LIN {X 0,Y 118.356,Z 1035.076,A -85,B 0,C 180,E1 -26009.999,E2 -26009.999} C_VEL
LIN {X 0,Y 118.425,Z 1040.689,A -85,B 0,C 180,E1 -26012.55,E2 -26012.55} C_VEL
LIN {X 0,Y 118.079,Z 1046.655,A -85,B 0,C 180,E1 -26015.978,E2 -26015.978} C_VEL
LIN {X 0,Y 117.481,Z 1052.345,A -85,B 0,C 180,E1 -26020.338,E2 -26020.338} C_VEL
LIN {X 0,Y 117.718,Z 1057.941,A -85,B 0,C 180,E1 -26025.528,E2 -26025.528} C_VEL
LIN {X 0,Y 119.258,Z 1062.55,A -85,B 0,C 180,E1 -26030.706,E2 -26030.706} C_VEL
LIN {X 0,Y 122.138,Z 1066.32,A -85,B 0,C 180,E1 -26035.566,E2 -26035.566} C_VEL
LIN {X 0,Y 126.034,Z 1069.156,A -85,B 0,C 180,E1 -26040.123,E2 -26040.123} C_VEL
LIN {X 0,Y 129.271,Z 1070.735,A -85,B 0,C 180,E1 -26042.933,E2 -26042.933} C_VEL
LIN {X 0,Y 137.158,Z 1072.698,A -85,B 0,C 180,E1 -26047.943,E2 -26047.943} C_VEL
LIN {X 0,Y 141.648,Z 1073.261,A -85,B 0,C 180,E1 -26050.166,E2 -26050.166} C_VEL
LIN {X 0,Y 151.624,Z 1073.236,A -85,B 0,C 180,E1 -26054.048,E2 -26054.048} C_VEL
LIN {X 0,Y 157.044,Z 1072.693,A -85,B 0,C 180,E1 -26055.727,E2 -26055.727} C_VEL
LIN {X 0,Y 157.853,Z 1072.521,A -85,B 0,C 180,E1 -26056.542,E2 -26056.542} C_VEL
LIN {X 0,Y 150.11,Z 1072.526,A -85,B 0,C 180,E1 -26059.047,E2 -26059.047} C_VEL
LIN {X 0,Y 142.602,Z 1071.645,A -85,B 0,C 180,E1 -26062.049,E2 -26062.049} C_VEL
LIN {X 0,Y 135.958,Z 1069.937,A -85,B 0,C 180,E1 -26065.348,E2 -26065.348} C_VEL
LIN {X 0,Y 130,Z 1067.367,A -85,B 0,C 180,E1 -26069.099,E2 -26069.099} C_VEL
LIN {X 0,Y 124.977,Z 1063.891,A -85,B 0,C 180,E1 -26073.266,E2 -26073.266} C_VEL
LIN {X 0,Y 121.04,Z 1059.399,A -85,B 0,C 180,E1 -26078.008,E2 -26078.008} C_VEL
LIN {X 0,Y 117.924,Z 1053.086,A -85,B 0,C 180,E1 -26083.593,E2 -26083.593} C_VEL
LIN {X 0,Y 116.582,Z 1047.62,A -85,B 0,C 180,E1 -26087.821,E2 -26087.821} C_VEL
LIN {X 0,Y 116.174,Z 1041.128,A -85,B 0,C 180,E1 -26092.179,E2 -26092.179} C_VEL
LIN {X 0,Y 116.121,Z 1034.894,A -85,B 0,C 180,E1 -26095.709,E2 -26095.709} C_VEL
LIN {X 0,Y 115.59,Z 1030.657,A -85,B 0,C 180,E1 -26097.651,E2 -26097.651} C_VEL
LIN {X 0,Y 114.297,Z 1025.939,A -85,B 0,C 180,E1 -26099.273,E2 -26099.273} C_VEL
LIN {X 0,Y 110.803,Z 1013.931,A -85,B 0,C 180,E1 -26102.592,E2 -26102.592} C_VEL
LIN {X 0,Y 110.37,Z 1008.52,A -85,B 0,C 180,E1 -26104.089,E2 -26104.089} C_VEL
LIN {X 0,Y 110.83,Z 996.455,A -85,B 0,C 180,E1 -26107.059,E2 -26107.059} C_VEL
LIN {X 0,Y 111.232,Z 984.797,A -85,B 0,C 180,E1 -26109.205,E2 -26109.205} C_VEL
LIN {X 0,Y 111.564,Z 944.315,A -85,B 0,C 180,E1 -26114.869,E2 -26114.869} C_VEL
LIN {X 0,Y 111.563,Z 935.848,A -85,B 0,C 180,E1 -26115.986,E2 -26115.986} C_VEL
LIN {X 0,Y 109.071,Z 921.711,A -85,B 0,C 180,E1 -26117.593,E2 -26117.593} C_VEL
LIN {X 0,Y 107.833,Z 921.864,A -85,B 0,C 180,E1 -26127.146,E2 -26127.146} C_VEL
LIN {X 0,Y 107.78,Z 921.869,A -85,B 0,C 180,E1 -26132.039,E2 -26132.039} C_VEL
LIN {X 0,Y 107.684,Z 921.876,A -85,B 0,C 180,E1 -26138.448,E2 -26138.448} C_VEL
LIN {X 0,Y 107.671,Z 921.883,A -85,B 0,C 180,E1 -26145.893,E2 -26145.893} C_VEL
LIN {X 0,Y 107.685,Z 921.882,A -85,B 0,C 180,E1 -26151.555,E2 -26151.555} C_VEL
LIN {X 0,Y 107.793,Z 921.862,A -85,B 0,C 180,E1 -26158.562,E2 -26158.562} C_VEL
LIN {X 0,Y 107.882,Z 921.851,A -85,B 0,C 180,E1 -26166.992,E2 -26166.992} C_VEL
LIN {X 0,Y 107.973,Z 921.842,A -85,B 0,C 180,E1 -26174.909,E2 -26174.909} C_VEL
LIN {X 0,Y 108.23,Z 921.813,A -85,B 0,C 180,E1 -26178.767,E2 -26178.767} C_VEL
LIN {X 0,Y 108.291,Z 921.806,A -85,B 0,C 180,E1 -26182.543,E2 -26182.543} C_VEL
LIN {X 0,Y 108.876,Z 921.737,A -85,B 0,C 180,E1 -26190.001,E2 -26190.001} C_VEL
LIN {X 0,Y 108.291,Z 921.806,A -85,B 0,C 180,E1 -26197.459,E2 -26197.459} C_VEL
LIN {X 0,Y 108.142,Z 921.819,A -85,B 0,C 180,E1 -26202.874,E2 -26202.874} C_VEL
LIN {X 0,Y 107.863,Z 921.862,A -85,B 0,C 180,E1 -26209.014,E2 -26209.014} C_VEL
LIN {X 0,Y 107.806,Z 921.862,A -85,B 0,C 180,E1 -26214.117,E2 -26214.117} C_VEL
LIN {X 0,Y 107.776,Z 921.863,A -85,B 0,C 180,E1 -26222.032,E2 -26222.032} C_VEL
LIN {X 0,Y 107.687,Z 921.882,A -85,B 0,C 180,E1 -26228.446,E2 -26228.446} C_VEL
LIN {X 0,Y 107.673,Z 921.886,A -85,B 0,C 180,E1 -26235.89,E2 -26235.89} C_VEL
LIN {X 0,Y 107.686,Z 921.876,A -85,B 0,C 180,E1 -26241.553,E2 -26241.553} C_VEL
LIN {X 0,Y 107.787,Z 921.865,A -85,B 0,C 180,E1 -26248.557,E2 -26248.557} C_VEL
LIN {X 0,Y 107.869,Z 921.857,A -85,B 0,C 180,E1 -26256.986,E2 -26256.986} C_VEL
LIN {X 0,Y 107.863,Z 921.856,A -85,B 0,C 180,E1 -26260.985,E2 -26260.985} C_VEL
LIN {X 0,Y 108.209,Z 921.809,A -85,B 0,C 180,E1 -26268.763,E2 -26268.763} C_VEL
LIN {X 0,Y 108.289,Z 921.808,A -85,B 0,C 180,E1 -26272.54,E2 -26272.54} C_VEL
LIN {X 0,Y 108.873,Z 921.732,A -85,B 0,C 180,E1 -26279.998,E2 -26279.998} C_VEL
LIN {X 0,Y 108.284,Z 921.801,A -85,B 0,C 180,E1 -26287.457,E2 -26287.457} C_VEL
LIN {X 0,Y 108.138,Z 921.826,A -85,B 0,C 180,E1 -26292.87,E2 -26292.87} C_VEL
LIN {X 0,Y 107.861,Z 921.86,A -85,B 0,C 180,E1 -26299.012,E2 -26299.012} C_VEL
LIN {X 0,Y 107.802,Z 921.864,A -85,B 0,C 180,E1 -26304.115,E2 -26304.115} C_VEL
LIN {X 0,Y 107.772,Z 921.87,A -85,B 0,C 180,E1 -26312.031,E2 -26312.031} C_VEL
LIN {X 0,Y 107.683,Z 921.883,A -85,B 0,C 180,E1 -26318.445,E2 -26318.445} C_VEL
LIN {X 0,Y 107.668,Z 921.882,A -85,B 0,C 180,E1 -26325.889,E2 -26325.889} C_VEL
LIN {X 0,Y 107.69,Z 921.879,A -85,B 0,C 180,E1 -26331.546,E2 -26331.546} C_VEL
LIN {X 0,Y 108.007,Z 921.843,A -85,B 0,C 180,E1 -26338.629,E2 -26338.629} C_VEL
LIN {X 0,Y 108.535,Z 921.78,A -85,B 0,C 180,E1 -26345.029,E2 -26345.029} C_VEL
LIN {X 0,Y 108.52,Z 921.977,A -85,B 0,C 180,E1 -26351.306,E2 -26351.306} C_VEL
LIN {X 0,Y 109.506,Z 943.925,A -85,B 0,C 180,E1 -26354.093,E2 -26354.093} C_VEL
LIN {X 0,Y 111.954,Z 966.951,A -85,B 0,C 180,E1 -26356.846,E2 -26356.846} C_VEL
LIN {X 0,Y 112.053,Z 995.999,A -85,B 0,C 180,E1 -26360.978,E2 -26360.978} C_VEL
LIN {X 0,Y 111.956,Z 1007.75,A -85,B 0,C 180,E1 -26363.24,E2 -26363.24} C_VEL
LIN {X 0,Y 111.912,Z 1018.14,A -85,B 0,C 180,E1 -26365.948,E2 -26365.948} C_VEL
LIN {X 0,Y 111.98,Z 1027.568,A -85,B 0,C 180,E1 -26369.1,E2 -26369.1} C_VEL
LIN {X 0,Y 112.088,Z 1034.186,A -85,B 0,C 180,E1 -26371.796,E2 -26371.796} C_VEL
LIN {X 0,Y 112.177,Z 1039.691,A -85,B 0,C 180,E1 -26374.491,E2 -26374.491} C_VEL
LIN {X 0,Y 111.753,Z 1045.35,A -85,B 0,C 180,E1 -26378.134,E2 -26378.134} C_VEL
LIN {X 0,Y 111.322,Z 1051.047,A -85,B 0,C 180,E1 -26382.765,E2 -26382.765} C_VEL
LIN {X 0,Y 112.15,Z 1057.246,A -85,B 0,C 180,E1 -26389.015,E2 -26389.015} C_VEL
LIN {X 0,Y 114.029,Z 1061.308,A -85,B 0,C 180,E1 -26393.616,E2 -26393.616} C_VEL
LIN {X 0,Y 117.42,Z 1065.087,A -85,B 0,C 180,E1 -26398.608,E2 -26398.608} C_VEL
LIN {X 0,Y 120.205,Z 1067.17,A -85,B 0,C 180,E1 -26401.749,E2 -26401.749} C_VEL
LIN {X 0,Y 127.45,Z 1070.367,A -85,B 0,C 180,E1 -26407.342,E2 -26407.342} C_VEL
LIN {X 0,Y 136.354,Z 1072.23,A -85,B 0,C 180,E1 -26412.07,E2 -26412.07} C_VEL
LIN {X 0,Y 141.307,Z 1072.763,A -85,B 0,C 180,E1 -26414.13,E2 -26414.13} C_VEL
LIN {X 0,Y 146.601,Z 1072.841,A -85,B 0,C 180,E1 -26415.979,E2 -26415.979} C_VEL
LIN {X 0,Y 144.811,Z 1072.568,A -85,B 0,C 180,E1 -26417.201,E2 -26417.201} C_VEL
LIN {X 0,Y 134.801,Z 1070.653,A -85,B 0,C 180,E1 -26421.273,E2 -26421.273} C_VEL
LIN {X 0,Y 126.016,Z 1067.11,A -85,B 0,C 180,E1 -26426.104,E2 -26426.104} C_VEL
LIN {X 0,Y 120.483,Z 1063.528,A -85,B 0,C 180,E1 -26430.278,E2 -26430.278} C_VEL
LIN {X 0,Y 116.099,Z 1059.034,A -85,B 0,C 180,E1 -26434.931,E2 -26434.931} C_VEL
LIN {X 0,Y 113.167,Z 1054.345,A -85,B 0,C 180,E1 -26439.358,E2 -26439.358} C_VEL
LIN {X 0,Y 110.941,Z 1048.163,A -85,B 0,C 180,E1 -26444.383,E2 -26444.383} C_VEL
LIN {X 0,Y 109.917,Z 1040.561,A -85,B 0,C 180,E1 -26449.875,E2 -26449.875} C_VEL
LIN {X 0,Y 109.813,Z 1032.534,A -85,B 0,C 180,E1 -26454.6,E2 -26454.6} C_VEL
LIN {X 0,Y 109.86,Z 1024.026,A -85,B 0,C 180,E1 -26458.627,E2 -26458.627} C_VEL
LIN {X 0,Y 110.115,Z 1014.241,A -85,B 0,C 180,E1 -26462.288,E2 -26462.288} C_VEL
LIN {X 0,Y 110.37,Z 1008.52,A -85,B 0,C 180,E1 -26464.089,E2 -26464.089} C_VEL
LIN {X 0,Y 109.99,Z 1003.267,A -85,B 0,C 180,E1 -26465.388,E2 -26465.388} C_VEL
LIN {X 0,Y 108.798,Z 997.812,A -85,B 0,C 180,E1 -26466.343,E2 -26466.343} C_VEL
LIN {X 0,Y 104.989,Z 982.527,A -85,B 0,C 180,E1 -26468.19,E2 -26468.19} C_VEL
LIN {X 0,Y 104.586,Z 978.592,A -85,B 0,C 180,E1 -26468.697,E2 -26468.697} C_VEL
LIN {X 0,Y 104.815,Z 939.202,A -85,B 0,C 180,E1 -26474.565,E2 -26474.565} C_VEL
LIN {X 0,Y 104.403,Z 933.942,A -85,B 0,C 180,E1 -26475.247,E2 -26475.247} C_VEL
LIN {X 0,Y 102.249,Z 922.562,A -85,B 0,C 180,E1 -26476.614,E2 -26476.614} C_VEL
LIN {X 0,Y 100.884,Z 922.732,A -85,B 0,C 180,E1 -26485.092,E2 -26485.092} C_VEL
LIN {X 0,Y 100.689,Z 922.753,A -85,B 0,C 180,E1 -26493.114,E2 -26493.114} C_VEL
LIN {X 0,Y 100.635,Z 922.753,A -85,B 0,C 180,E1 -26499.809,E2 -26499.809} C_VEL
LIN {X 0,Y 100.642,Z 922.759,A -85,B 0,C 180,E1 -26505.709,E2 -26505.709} C_VEL
LIN {X 0,Y 100.623,Z 922.762,A -85,B 0,C 180,E1 -26511.054,E2 -26511.054} C_VEL
LIN {X 0,Y 100.69,Z 922.746,A -85,B 0,C 180,E1 -26516.889,E2 -26516.889} C_VEL
LIN {X 0,Y 100.737,Z 922.744,A -85,B 0,C 180,E1 -26525.093,E2 -26525.093} C_VEL
LIN {X 0,Y 100.785,Z 922.742,A -85,B 0,C 180,E1 -26529.595,E2 -26529.595} C_VEL
LIN {X 0,Y 101.129,Z 922.696,A -85,B 0,C 180,E1 -26537.967,E2 -26537.967} C_VEL
LIN {X 0,Y 101.229,Z 922.687,A -85,B 0,C 180,E1 -26542.019,E2 -26542.019} C_VEL
LIN {X 0,Y 101.807,Z 922.617,A -85,B 0,C 180,E1 -26550.001,E2 -26550.001} C_VEL
LIN {X 0,Y 101.228,Z 922.687,A -85,B 0,C 180,E1 -26557.982,E2 -26557.982} C_VEL
LIN {X 0,Y 101.054,Z 922.701,A -85,B 0,C 180,E1 -26563.171,E2 -26563.171} C_VEL
LIN {X 0,Y 100.777,Z 922.743,A -85,B 0,C 180,E1 -26570.408,E2 -26570.408} C_VEL
LIN {X 0,Y 100.721,Z 922.746,A -85,B 0,C 180,E1 -26574.887,E2 -26574.887} C_VEL
LIN {X 0,Y 100.688,Z 922.747,A -85,B 0,C 180,E1 -26583.109,E2 -26583.109} C_VEL
LIN {X 0,Y 100.638,Z 922.756,A -85,B 0,C 180,E1 -26589.806,E2 -26589.806} C_VEL
LIN {X 0,Y 100.644,Z 922.761,A -85,B 0,C 180,E1 -26595.706,E2 -26595.706} C_VEL
LIN {X 0,Y 100.624,Z 922.754,A -85,B 0,C 180,E1 -26601.051,E2 -26601.051} C_VEL
LIN {X 0,Y 100.688,Z 922.754,A -85,B 0,C 180,E1 -26606.889,E2 -26606.889} C_VEL
LIN {X 0,Y 100.745,Z 922.748,A -85,B 0,C 180,E1 -26615.254,E2 -26615.254} C_VEL
LIN {X 0,Y 100.778,Z 922.736,A -85,B 0,C 180,E1 -26619.591,E2 -26619.591} C_VEL
LIN {X 0,Y 101.118,Z 922.692,A -85,B 0,C 180,E1 -26627.963,E2 -26627.963} C_VEL
LIN {X 0,Y 101.224,Z 922.689,A -85,B 0,C 180,E1 -26632.016,E2 -26632.016} C_VEL
LIN {X 0,Y 101.805,Z 922.613,A -85,B 0,C 180,E1 -26639.998,E2 -26639.998} C_VEL
LIN {X 0,Y 101.219,Z 922.681,A -85,B 0,C 180,E1 -26647.98,E2 -26647.98} C_VEL
LIN {X 0,Y 101.051,Z 922.708,A -85,B 0,C 180,E1 -26653.169,E2 -26653.169} C_VEL
LIN {X 0,Y 100.774,Z 922.744,A -85,B 0,C 180,E1 -26660.406,E2 -26660.406} C_VEL
LIN {X 0,Y 100.717,Z 922.743,A -85,B 0,C 180,E1 -26664.886,E2 -26664.886} C_VEL
LIN {X 0,Y 100.684,Z 922.75,A -85,B 0,C 180,E1 -26673.108,E2 -26673.108} C_VEL
LIN {X 0,Y 100.634,Z 922.762,A -85,B 0,C 180,E1 -26679.805,E2 -26679.805} C_VEL
LIN {X 0,Y 100.639,Z 922.756,A -85,B 0,C 180,E1 -26685.705,E2 -26685.705} C_VEL
LIN {X 0,Y 100.627,Z 922.759,A -85,B 0,C 180,E1 -26691.054,E2 -26691.054} C_VEL
LIN {X 0,Y 100.793,Z 922.743,A -85,B 0,C 180,E1 -26696.793,E2 -26696.793} C_VEL
LIN {X 0,Y 101.378,Z 922.668,A -85,B 0,C 180,E1 -26704.315,E2 -26704.315} C_VEL
LIN {X 0,Y 101.61,Z 922.642,A -85,B 0,C 180,E1 -26712.255,E2 -26712.255} C_VEL
LIN {X 0,Y 102.806,Z 945.114,A -85,B 0,C 180,E1 -26715.335,E2 -26715.335} C_VEL
LIN {X 0,Y 105.267,Z 967.587,A -85,B 0,C 180,E1 -26718.201,E2 -26718.201} C_VEL
LIN {X 0,Y 105.553,Z 996.226,A -85,B 0,C 180,E1 -26722.587,E2 -26722.587} C_VEL
LIN {X 0,Y 105.558,Z 1008.784,A -85,B 0,C 180,E1 -26725.225,E2 -26725.225} C_VEL
LIN {X 0,Y 105.625,Z 1020.086,A -85,B 0,C 180,E1 -26728.568,E2 -26728.568} C_VEL
LIN {X 0,Y 105.891,Z 1028.857,A -85,B 0,C 180,E1 -26731.901,E2 -26731.901} C_VEL
LIN {X 0,Y 106.139,Z 1036.77,A -85,B 0,C 180,E1 -26735.701,E2 -26735.701} C_VEL
LIN {X 0,Y 105.886,Z 1041.269,A -85,B 0,C 180,E1 -26738.588,E2 -26738.588} C_VEL
LIN {X 0,Y 105.412,Z 1047.304,A -85,B 0,C 180,E1 -26743.494,E2 -26743.494} C_VEL
LIN {X 0,Y 106.318,Z 1054.567,A -85,B 0,C 180,E1 -26750.676,E2 -26750.676} C_VEL
LIN {X 0,Y 110.355,Z 1061.207,A -85,B 0,C 180,E1 -26758.531,E2 -26758.531} C_VEL
LIN {X 0,Y 114.566,Z 1064.808,A -85,B 0,C 180,E1 -26763.511,E2 -26763.511} C_VEL
LIN {X 0,Y 118.065,Z 1066.85,A -85,B 0,C 180,E1 -26766.531,E2 -26766.531} C_VEL
LIN {X 0,Y 126.486,Z 1069.936,A -85,B 0,C 180,E1 -26771.817,E2 -26771.817} C_VEL
LIN {X 0,Y 136.365,Z 1071.739,A -85,B 0,C 180,E1 -26776.181,E2 -26776.181} C_VEL
LIN {X 0,Y 132.956,Z 1070.914,A -85,B 0,C 180,E1 -26777.734,E2 -26777.734} C_VEL
LIN {X 0,Y 122.436,Z 1066.822,A -85,B 0,C 180,E1 -26782.937,E2 -26782.937} C_VEL
LIN {X 0,Y 116.375,Z 1063.037,A -85,B 0,C 180,E1 -26787.078,E2 -26787.078} C_VEL
LIN {X 0,Y 111.285,Z 1058.298,A -85,B 0,C 180,E1 -26791.936,E2 -26791.936} C_VEL
LIN {X 0,Y 107.022,Z 1051.645,A -85,B 0,C 180,E1 -26798.114,E2 -26798.114} C_VEL
LIN {X 0,Y 104.467,Z 1043.763,A -85,B 0,C 180,E1 -26804.391,E2 -26804.391} C_VEL
LIN {X 0,Y 103.735,Z 1035.281,A -85,B 0,C 180,E1 -26810.25,E2 -26810.25} C_VEL
LIN {X 0,Y 103.661,Z 1028.425,A -85,B 0,C 180,E1 -26814.165,E2 -26814.165} C_VEL
LIN {X 0,Y 103.678,Z 1019.9,A -85,B 0,C 180,E1 -26818.059,E2 -26818.059} C_VEL
LIN {X 0,Y 103.888,Z 1009.362,A -85,B 0,C 180,E1 -26821.94,E2 -26821.94} C_VEL
LIN {X 0,Y 104.223,Z 998.058,A -85,B 0,C 180,E1 -26825.079,E2 -26825.079} C_VEL
LIN {X 0,Y 104.551,Z 987.696,A -85,B 0,C 180,E1 -26827.243,E2 -26827.243} C_VEL
LIN {X 0,Y 104.586,Z 978.592,A -85,B 0,C 180,E1 -26828.697,E2 -26828.697} C_VEL
LIN {X 0,Y 103.841,Z 972.861,A -85,B 0,C 180,E1 -26829.409,E2 -26829.409} C_VEL
LIN {X 0,Y 98.573,Z 954.007,A -85,B 0,C 180,E1 -26831.225,E2 -26831.225} C_VEL
LIN {X 0,Y 97.979,Z 948.282,A -85,B 0,C 180,E1 -26832.006,E2 -26832.006} C_VEL
LIN {X 0,Y 97.787,Z 935.443,A -85,B 0,C 180,E1 -26833.957,E2 -26833.957} C_VEL
LIN {X 0,Y 95.48,Z 923.405,A -85,B 0,C 180,E1 -26835.453,E2 -26835.453} C_VEL
LIN {X 0,Y 93.708,Z 923.625,A -85,B 0,C 180,E1 -26846.746,E2 -26846.746} C_VEL
LIN {X 0,Y 93.585,Z 923.64,A -85,B 0,C 180,E1 -26854.304,E2 -26854.304} C_VEL
LIN {X 0,Y 93.529,Z 923.647,A -85,B 0,C 180,E1 -26862.557,E2 -26862.557} C_VEL
LIN {X 0,Y 93.532,Z 923.638,A -85,B 0,C 180,E1 -26868.715,E2 -26868.715} C_VEL
LIN {X 0,Y 93.586,Z 923.636,A -85,B 0,C 180,E1 -26875.7,E2 -26875.7} C_VEL
LIN {X 0,Y 93.646,Z 923.631,A -85,B 0,C 180,E1 -26884.24,E2 -26884.24} C_VEL
LIN {X 0,Y 93.657,Z 923.624,A -85,B 0,C 180,E1 -26887.964,E2 -26887.964} C_VEL
LIN {X 0,Y 94.019,Z 923.577,A -85,B 0,C 180,E1 -26897.042,E2 -26897.042} C_VEL
LIN {X 0,Y 94.16,Z 923.569,A -85,B 0,C 180,E1 -26901.416,E2 -26901.416} C_VEL
LIN {X 0,Y 94.739,Z 923.497,A -85,B 0,C 180,E1 -26910.001,E2 -26910.001} C_VEL
LIN {X 0,Y 94.16,Z 923.569,A -85,B 0,C 180,E1 -26918.586,E2 -26918.586} C_VEL
LIN {X 0,Y 93.962,Z 923.584,A -85,B 0,C 180,E1 -26923.496,E2 -26923.496} C_VEL
LIN {X 0,Y 93.646,Z 923.625,A -85,B 0,C 180,E1 -26932.04,E2 -26932.04} C_VEL
LIN {X 0,Y 93.591,Z 923.639,A -85,B 0,C 180,E1 -26936.78,E2 -26936.78} C_VEL
LIN {X 0,Y 93.586,Z 923.636,A -85,B 0,C 180,E1 -26944.299,E2 -26944.299} C_VEL
LIN {X 0,Y 93.531,Z 923.64,A -85,B 0,C 180,E1 -26952.554,E2 -26952.554} C_VEL
LIN {X 0,Y 93.534,Z 923.642,A -85,B 0,C 180,E1 -26958.712,E2 -26958.712} C_VEL
LIN {X 0,Y 93.585,Z 923.64,A -85,B 0,C 180,E1 -26965.699,E2 -26965.699} C_VEL
LIN {X 0,Y 93.644,Z 923.632,A -85,B 0,C 180,E1 -26974.239,E2 -26974.239} C_VEL
LIN {X 0,Y 93.653,Z 923.625,A -85,B 0,C 180,E1 -26977.96,E2 -26977.96} C_VEL
LIN {X 0,Y 94.018,Z 923.58,A -85,B 0,C 180,E1 -26987.039,E2 -26987.039} C_VEL
LIN {X 0,Y 94.135,Z 923.57,A -85,B 0,C 180,E1 -26991.411,E2 -26991.411} C_VEL
LIN {X 0,Y 94.737,Z 923.493,A -85,B 0,C 180,E1 -26999.998,E2 -26999.998} C_VEL
LIN {X 0,Y 94.131,Z 923.566,A -85,B 0,C 180,E1 -27008.586,E2 -27008.586} C_VEL
LIN {X 0,Y 93.959,Z 923.591,A -85,B 0,C 180,E1 -27013.494,E2 -27013.494} C_VEL
LIN {X 0,Y 93.643,Z 923.632,A -85,B 0,C 180,E1 -27022.038,E2 -27022.038} C_VEL
LIN {X 0,Y 93.587,Z 923.633,A -85,B 0,C 180,E1 -27026.779,E2 -27026.779} C_VEL
LIN {X 0,Y 93.582,Z 923.63,A -85,B 0,C 180,E1 -27034.298,E2 -27034.298} C_VEL
LIN {X 0,Y 93.526,Z 923.641,A -85,B 0,C 180,E1 -27042.553,E2 -27042.553} C_VEL
LIN {X 0,Y 93.532,Z 923.646,A -85,B 0,C 180,E1 -27048.709,E2 -27048.709} C_VEL
LIN {X 0,Y 93.655,Z 923.629,A -85,B 0,C 180,E1 -27055.632,E2 -27055.632} C_VEL
LIN {X 0,Y 94.206,Z 923.556,A -85,B 0,C 180,E1 -27063.534,E2 -27063.534} C_VEL
LIN {X 0,Y 94.314,Z 923.55,A -85,B 0,C 180,E1 -27068.124,E2 -27068.124} C_VEL
LIN {X 0,Y 94.794,Z 923.492,A -85,B 0,C 180,E1 -27073.436,E2 -27073.436} C_VEL
LIN {X 0,Y 96.131,Z 945.61,A -85,B 0,C 180,E1 -27076.686,E2 -27076.686} C_VEL
LIN {X 0,Y 98.642,Z 967.237,A -85,B 0,C 180,E1 -27079.609,E2 -27079.609} C_VEL
LIN {X 0,Y 99.15,Z 995.476,A -85,B 0,C 180,E1 -27084.253,E2 -27084.253} C_VEL
LIN {X 0,Y 99.307,Z 1007.466,A -85,B 0,C 180,E1 -27086.957,E2 -27086.957} C_VEL
LIN {X 0,Y 99.531,Z 1018.258,A -85,B 0,C 180,E1 -27090.32,E2 -27090.32} C_VEL
LIN {X 0,Y 99.883,Z 1026.452,A -85,B 0,C 180,E1 -27093.529,E2 -27093.529} C_VEL
LIN {X 0,Y 100.183,Z 1033.301,A -85,B 0,C 180,E1 -27096.848,E2 -27096.848} C_VEL
LIN {X 0,Y 99.959,Z 1038.433,A -85,B 0,C 180,E1 -27100.169,E2 -27100.169} C_VEL
LIN {X 0,Y 99.7,Z 1045.625,A -85,B 0,C 180,E1 -27106.377,E2 -27106.377} C_VEL
LIN {X 0,Y 100.786,Z 1051.611,A -85,B 0,C 180,E1 -27112.552,E2 -27112.552} C_VEL
LIN {X 0,Y 103.506,Z 1056.729,A -85,B 0,C 180,E1 -27118.378,E2 -27118.378} C_VEL
LIN {X 0,Y 107.553,Z 1060.954,A -85,B 0,C 180,E1 -27123.74,E2 -27123.74} C_VEL
LIN {X 0,Y 112.777,Z 1064.465,A -85,B 0,C 180,E1 -27128.548,E2 -27128.548} C_VEL
LIN {X 0,Y 116.911,Z 1066.461,A -85,B 0,C 180,E1 -27131.395,E2 -27131.395} C_VEL
LIN {X 0,Y 124.966,Z 1069.131,A -85,B 0,C 180,E1 -27135.675,E2 -27135.675} C_VEL
LIN {X 0,Y 125.191,Z 1069.057,A -85,B 0,C 180,E1 -27136.721,E2 -27136.721} C_VEL
LIN {X 0,Y 116.982,Z 1065.239,A -85,B 0,C 180,E1 -27140.892,E2 -27140.892} C_VEL
LIN {X 0,Y 110.708,Z 1061.033,A -85,B 0,C 180,E1 -27145.158,E2 -27145.158} C_VEL
LIN {X 0,Y 105.602,Z 1055.984,A -85,B 0,C 180,E1 -27150.057,E2 -27150.057} C_VEL
LIN {X 0,Y 101.72,Z 1049.995,A -85,B 0,C 180,E1 -27155.511,E2 -27155.511} C_VEL
LIN {X 0,Y 99.018,Z 1042.801,A -85,B 0,C 180,E1 -27161.376,E2 -27161.376} C_VEL
LIN {X 0,Y 97.939,Z 1035.838,A -85,B 0,C 180,E1 -27166.515,E2 -27166.515} C_VEL
LIN {X 0,Y 97.656,Z 1029.281,A -85,B 0,C 180,E1 -27170.683,E2 -27170.683} C_VEL
LIN {X 0,Y 97.563,Z 1022.495,A -85,B 0,C 180,E1 -27174.317,E2 -27174.317} C_VEL
LIN {X 0,Y 97.56,Z 1014.148,A -85,B 0,C 180,E1 -27177.938,E2 -27177.938} C_VEL
LIN {X 0,Y 97.702,Z 1003.575,A -85,B 0,C 180,E1 -27181.548,E2 -27181.548} C_VEL
LIN {X 0,Y 97.991,Z 991.655,A -85,B 0,C 180,E1 -27184.63,E2 -27184.63} C_VEL
LIN {X 0,Y 98.148,Z 980.058,A -85,B 0,C 180,E1 -27186.813,E2 -27186.813} C_VEL
LIN {X 0,Y 97.979,Z 948.282,A -85,B 0,C 180,E1 -27192.006,E2 -27192.006} C_VEL
LIN {X 0,Y 97.305,Z 944.486,A -85,B 0,C 180,E1 -27192.478,E2 -27192.478} C_VEL
LIN {X 0,Y 94.335,Z 938.527,A -85,B 0,C 180,E1 -27192.8,E2 -27192.8} C_VEL
LIN {X 0,Y 90.979,Z 932.584,A -85,B 0,C 180,E1 -27193.04,E2 -27193.04} C_VEL
LIN {X 0,Y 89.737,Z 928.775,A -85,B 0,C 180,E1 -27193.406,E2 -27193.406} C_VEL
LIN {X 0,Y 88.817,Z 924.232,A -85,B 0,C 180,E1 -27194.044,E2 -27194.044} C_VEL
LIN {X 0,Y 86.54,Z 924.509,A -85,B 0,C 180,E1 -27209.164,E2 -27209.164} C_VEL
LIN {X 0,Y 86.503,Z 924.521,A -85,B 0,C 180,E1 -27215.665,E2 -27215.665} C_VEL
LIN {X 0,Y 86.473,Z 924.525,A -85,B 0,C 180,E1 -27222.992,E2 -27222.992} C_VEL
LIN {X 0,Y 86.455,Z 924.52,A -85,B 0,C 180,E1 -27229.435,E2 -27229.435} C_VEL
LIN {X 0,Y 86.529,Z 924.516,A -85,B 0,C 180,E1 -27235.352,E2 -27235.352} C_VEL
LIN {X 0,Y 86.569,Z 924.513,A -85,B 0,C 180,E1 -27243.261,E2 -27243.261} C_VEL
LIN {X 0,Y 86.603,Z 924.51,A -85,B 0,C 180,E1 -27251.059,E2 -27251.059} C_VEL
LIN {X 0,Y 86.866,Z 924.467,A -85,B 0,C 180,E1 -27256.147,E2 -27256.147} C_VEL
LIN {X 0,Y 87.064,Z 924.452,A -85,B 0,C 180,E1 -27260.71,E2 -27260.71} C_VEL
LIN {X 0,Y 87.672,Z 924.378,A -85,B 0,C 180,E1 -27270.001,E2 -27270.001} C_VEL
LIN {X 0,Y 87.063,Z 924.452,A -85,B 0,C 180,E1 -27279.292,E2 -27279.292} C_VEL
LIN {X 0,Y 86.863,Z 924.467,A -85,B 0,C 180,E1 -27284.048,E2 -27284.048} C_VEL
LIN {X 0,Y 86.597,Z 924.511,A -85,B 0,C 180,E1 -27288.944,E2 -27288.944} C_VEL
LIN {X 0,Y 86.559,Z 924.514,A -85,B 0,C 180,E1 -27296.726,E2 -27296.726} C_VEL
LIN {X 0,Y 86.505,Z 924.521,A -85,B 0,C 180,E1 -27305.661,E2 -27305.661} C_VEL
LIN {X 0,Y 86.475,Z 924.52,A -85,B 0,C 180,E1 -27312.989,E2 -27312.989} C_VEL
LIN {X 0,Y 86.456,Z 924.521,A -85,B 0,C 180,E1 -27319.431,E2 -27319.431} C_VEL
LIN {X 0,Y 86.529,Z 924.519,A -85,B 0,C 180,E1 -27325.348,E2 -27325.348} C_VEL
LIN {X 0,Y 86.565,Z 924.514,A -85,B 0,C 180,E1 -27333.263,E2 -27333.263} C_VEL
LIN {X 0,Y 86.598,Z 924.505,A -85,B 0,C 180,E1 -27341.055,E2 -27341.055} C_VEL
LIN {X 0,Y 86.864,Z 924.474,A -85,B 0,C 180,E1 -27346.147,E2 -27346.147} C_VEL
LIN {X 0,Y 87.028,Z 924.454,A -85,B 0,C 180,E1 -27350.703,E2 -27350.703} C_VEL
LIN {X 0,Y 87.669,Z 924.373,A -85,B 0,C 180,E1 -27359.998,E2 -27359.998} C_VEL
LIN {X 0,Y 87.025,Z 924.455,A -85,B 0,C 180,E1 -27369.293,E2 -27369.293} C_VEL
LIN {X 0,Y 86.86,Z 924.474,A -85,B 0,C 180,E1 -27374.046,E2 -27374.046} C_VEL
LIN {X 0,Y 86.594,Z 924.509,A -85,B 0,C 180,E1 -27378.942,E2 -27378.942} C_VEL
LIN {X 0,Y 86.555,Z 924.509,A -85,B 0,C 180,E1 -27386.724,E2 -27386.724} C_VEL
LIN {X 0,Y 86.501,Z 924.514,A -85,B 0,C 180,E1 -27395.659,E2 -27395.659} C_VEL
LIN {X 0,Y 86.45,Z 924.521,A -85,B 0,C 180,E1 -27402.973,E2 -27402.973} C_VEL
LIN {X 0,Y 86.458,Z 924.527,A -85,B 0,C 180,E1 -27409.434,E2 -27409.434} C_VEL
LIN {X 0,Y 86.59,Z 924.509,A -85,B 0,C 180,E1 -27415.378,E2 -27415.378} C_VEL
LIN {X 0,Y 87.021,Z 924.448,A -85,B 0,C 180,E1 -27422.667,E2 -27422.667} C_VEL
LIN {X 0,Y 87.151,Z 924.443,A -85,B 0,C 180,E1 -27426.22,E2 -27426.22} C_VEL
LIN {X 0,Y 88.055,Z 924.493,A -85,B 0,C 180,E1 -27434.932,E2 -27434.932} C_VEL
LIN {X 0,Y 89.7,Z 947.203,A -85,B 0,C 180,E1 -27438.489,E2 -27438.489} C_VEL
LIN {X 0,Y 92.185,Z 967.673,A -85,B 0,C 180,E1 -27441.444,E2 -27441.444} C_VEL
LIN {X 0,Y 92.952,Z 995.045,A -85,B 0,C 180,E1 -27446.342,E2 -27446.342} C_VEL
LIN {X 0,Y 93.225,Z 1005.858,A -85,B 0,C 180,E1 -27448.919,E2 -27448.919} C_VEL
LIN {X 0,Y 93.538,Z 1016.48,A -85,B 0,C 180,E1 -27452.323,E2 -27452.323} C_VEL
LIN {X 0,Y 94.005,Z 1024.301,A -85,B 0,C 180,E1 -27455.499,E2 -27455.499} C_VEL
LIN {X 0,Y 94.415,Z 1030.372,A -85,B 0,C 180,E1 -27458.561,E2 -27458.561} C_VEL
LIN {X 0,Y 94.301,Z 1035.149,A -85,B 0,C 180,E1 -27461.85,E2 -27461.85} C_VEL
LIN {X 0,Y 94.139,Z 1042.704,A -85,B 0,C 180,E1 -27468.498,E2 -27468.498} C_VEL
LIN {X 0,Y 95.976,Z 1049.844,A -85,B 0,C 180,E1 -27476.062,E2 -27476.062} C_VEL
LIN {X 0,Y 98.975,Z 1054.63,A -85,B 0,C 180,E1 -27481.563,E2 -27481.563} C_VEL
LIN {X 0,Y 105.758,Z 1060.587,A -85,B 0,C 180,E1 -27489.146,E2 -27489.146} C_VEL
LIN {X 0,Y 112.017,Z 1063.999,A -85,B 0,C 180,E1 -27493.641,E2 -27493.641} C_VEL
LIN {X 0,Y 114.191,Z 1064.948,A -85,B 0,C 180,E1 -27494.914,E2 -27494.914} C_VEL
LIN {X 0,Y 115.347,Z 1065.295,A -85,B 0,C 180,E1 -27496.714,E2 -27496.714} C_VEL
LIN {X 0,Y 107.32,Z 1060.206,A -85,B 0,C 180,E1 -27501.531,E2 -27501.531} C_VEL
LIN {X 0,Y 101.596,Z 1055.017,A -85,B 0,C 180,E1 -27506.401,E2 -27506.401} C_VEL
LIN {X 0,Y 96.628,Z 1048.001,A -85,B 0,C 180,E1 -27512.812,E2 -27512.812} C_VEL
LIN {X 0,Y 93.973,Z 1041.729,A -85,B 0,C 180,E1 -27518.044,E2 -27518.044} C_VEL
LIN {X 0,Y 92.069,Z 1031.637,A -85,B 0,C 180,E1 -27525.638,E2 -27525.638} C_VEL
LIN {X 0,Y 91.782,Z 1023.515,A -85,B 0,C 180,E1 -27530.637,E2 -27530.637} C_VEL
LIN {X 0,Y 91.589,Z 1014.352,A -85,B 0,C 180,E1 -27535.05,E2 -27535.05} C_VEL
LIN {X 0,Y 91.58,Z 1004.63,A -85,B 0,C 180,E1 -27538.793,E2 -27538.793} C_VEL
LIN {X 0,Y 91.671,Z 992.875,A -85,B 0,C 180,E1 -27542.199,E2 -27542.199} C_VEL
LIN {X 0,Y 91.874,Z 980.598,A -85,B 0,C 180,E1 -27544.757,E2 -27544.757} C_VEL
LIN {X 0,Y 91.266,Z 936.91,A -85,B 0,C 180,E1 -27552.369,E2 -27552.369} C_VEL
LIN {X 0,Y 89.737,Z 928.775,A -85,B 0,C 180,E1 -27553.406,E2 -27553.406} C_VEL
LIN {X 0,Y 88.951,Z 926.803,A -85,B 0,C 180,E1 -27554.115,E2 -27554.115} C_VEL
LIN {X 0,Y 87.369,Z 925.292,A -85,B 0,C 180,E1 -27555.762,E2 -27555.762} C_VEL
LIN {X 0,Y 85.157,Z 924.745,A -85,B 0,C 180,E1 -27558.468,E2 -27558.468} C_VEL
LIN {X 0,Y 80.592,Z 925.298,A -85,B 0,C 180,E1 -27566.993,E2 -27566.993} C_VEL
LIN {X 0,Y 79.331,Z 925.403,A -85,B 0,C 180,E1 -27573.597,E2 -27573.597} C_VEL
LIN {X 0,Y 79.363,Z 925.403,A -85,B 0,C 180,E1 -27578.311,E2 -27578.311} C_VEL
LIN {X 0,Y 79.386,Z 925.408,A -85,B 0,C 180,E1 -27585.095,E2 -27585.095} C_VEL
LIN {X 0,Y 79.385,Z 925.409,A -85,B 0,C 180,E1 -27592.827,E2 -27592.827} C_VEL
LIN {X 0,Y 79.373,Z 925.4,A -85,B 0,C 180,E1 -27597.91,E2 -27597.91} C_VEL
LIN {X 0,Y 79.51,Z 925.392,A -85,B 0,C 180,E1 -27603.772,E2 -27603.772} C_VEL
LIN {X 0,Y 79.481,Z 925.393,A -85,B 0,C 180,E1 -27609.287,E2 -27609.287} C_VEL
LIN {X 0,Y 79.79,Z 925.348,A -85,B 0,C 180,E1 -27615.681,E2 -27615.681} C_VEL
LIN {X 0,Y 79.939,Z 925.34,A -85,B 0,C 180,E1 -27619.874,E2 -27619.874} C_VEL
LIN {X 0,Y 80.604,Z 925.258,A -85,B 0,C 180,E1 -27630.001,E2 -27630.001} C_VEL
LIN {X 0,Y 79.938,Z 925.34,A -85,B 0,C 180,E1 -27640.128,E2 -27640.128} C_VEL
LIN {X 0,Y 79.69,Z 925.364,A -85,B 0,C 180,E1 -27645.343,E2 -27645.343} C_VEL
LIN {X 0,Y 79.474,Z 925.394,A -85,B 0,C 180,E1 -27650.717,E2 -27650.717} C_VEL
LIN {X 0,Y 79.462,Z 925.399,A -85,B 0,C 180,E1 -27657.811,E2 -27657.811} C_VEL
LIN {X 0,Y 79.37,Z 925.4,A -85,B 0,C 180,E1 -27662.094,E2 -27662.094} C_VEL
LIN {X 0,Y 79.365,Z 925.41,A -85,B 0,C 180,E1 -27668.308,E2 -27668.308} C_VEL
LIN {X 0,Y 79.388,Z 925.408,A -85,B 0,C 180,E1 -27675.092,E2 -27675.092} C_VEL
LIN {X 0,Y 79.386,Z 925.404,A -85,B 0,C 180,E1 -27682.825,E2 -27682.825} C_VEL
LIN {X 0,Y 79.371,Z 925.406,A -85,B 0,C 180,E1 -27687.905,E2 -27687.905} C_VEL
LIN {X 0,Y 79.506,Z 925.393,A -85,B 0,C 180,E1 -27693.767,E2 -27693.767} C_VEL
LIN {X 0,Y 79.477,Z 925.388,A -85,B 0,C 180,E1 -27699.283,E2 -27699.283} C_VEL
LIN {X 0,Y 79.788,Z 925.356,A -85,B 0,C 180,E1 -27705.683,E2 -27705.683} C_VEL
LIN {X 0,Y 79.913,Z 925.335,A -85,B 0,C 180,E1 -27709.867,E2 -27709.867} C_VEL
LIN {X 0,Y 80.601,Z 925.253,A -85,B 0,C 180,E1 -27719.998,E2 -27719.998} C_VEL
LIN {X 0,Y 79.91,Z 925.342,A -85,B 0,C 180,E1 -27730.129,E2 -27730.129} C_VEL
LIN {X 0,Y 79.687,Z 925.362,A -85,B 0,C 180,E1 -27735.34,E2 -27735.34} C_VEL
LIN {X 0,Y 79.471,Z 925.399,A -85,B 0,C 180,E1 -27740.714,E2 -27740.714} C_VEL
LIN {X 0,Y 79.458,Z 925.396,A -85,B 0,C 180,E1 -27747.808,E2 -27747.808} C_VEL
LIN {X 0,Y 79.366,Z 925.408,A -85,B 0,C 180,E1 -27752.091,E2 -27752.091} C_VEL
LIN {X 0,Y 79.361,Z 925.412,A -85,B 0,C 180,E1 -27758.306,E2 -27758.306} C_VEL
LIN {X 0,Y 79.381,Z 925.402,A -85,B 0,C 180,E1 -27765.092,E2 -27765.092} C_VEL
LIN {X 0,Y 79.41,Z 925.396,A -85,B 0,C 180,E1 -27772.796,E2 -27772.796} C_VEL
LIN {X 0,Y 79.868,Z 925.34,A -85,B 0,C 180,E1 -27781.632,E2 -27781.632} C_VEL
LIN {X 0,Y 80.187,Z 925.308,A -85,B 0,C 180,E1 -27789.476,E2 -27789.476} C_VEL
LIN {X 0,Y 81.42,Z 925.272,A -85,B 0,C 180,E1 -27796.744,E2 -27796.744} C_VEL
LIN {X 0,Y 83.439,Z 949.096,A -85,B 0,C 180,E1 -27800.712,E2 -27800.712} C_VEL
LIN {X 0,Y 85.857,Z 967.597,A -85,B 0,C 180,E1 -27803.543,E2 -27803.543} C_VEL
LIN {X 0,Y 86.88,Z 994.449,A -85,B 0,C 180,E1 -27808.695,E2 -27808.695} C_VEL
LIN {X 0,Y 87.311,Z 1004.175,A -85,B 0,C 180,E1 -27811.152,E2 -27811.152} C_VEL
LIN {X 0,Y 87.816,Z 1014.335,A -85,B 0,C 180,E1 -27814.59,E2 -27814.59} C_VEL
LIN {X 0,Y 88.54,Z 1023.502,A -85,B 0,C 180,E1 -27818.558,E2 -27818.558} C_VEL
LIN {X 0,Y 88.951,Z 1028.713,A -85,B 0,C 180,E1 -27821.444,E2 -27821.444} C_VEL
LIN {X 0,Y 88.72,Z 1032.912,A -85,B 0,C 180,E1 -27824.681,E2 -27824.681} C_VEL
LIN {X 0,Y 88.949,Z 1039.448,A -85,B 0,C 180,E1 -27830.827,E2 -27830.827} C_VEL
LIN {X 0,Y 90.681,Z 1045.909,A -85,B 0,C 180,E1 -27837.71,E2 -27837.71} C_VEL
LIN {X 0,Y 95.653,Z 1053.149,A -85,B 0,C 180,E1 -27846,E2 -27846} C_VEL
LIN {X 0,Y 102.898,Z 1058.857,A -85,B 0,C 180,E1 -27853.078,E2 -27853.078} C_VEL
LIN {X 0,Y 106.166,Z 1060.68,A -85,B 0,C 180,E1 -27855.312,E2 -27855.312} C_VEL
LIN {X 0,Y 106.828,Z 1060.983,A -85,B 0,C 180,E1 -27856.269,E2 -27856.269} C_VEL
LIN {X 0,Y 100.105,Z 1055.818,A -85,B 0,C 180,E1 -27860.815,E2 -27860.815} C_VEL
LIN {X 0,Y 95.382,Z 1050.984,A -85,B 0,C 180,E1 -27865.232,E2 -27865.232} C_VEL
LIN {X 0,Y 91.039,Z 1044.259,A -85,B 0,C 180,E1 -27871.154,E2 -27871.154} C_VEL
LIN {X 0,Y 87.897,Z 1036.308,A -85,B 0,C 180,E1 -27877.681,E2 -27877.681} C_VEL
LIN {X 0,Y 86.474,Z 1026.898,A -85,B 0,C 180,E1 -27884.686,E2 -27884.686} C_VEL
LIN {X 0,Y 85.98,Z 1018.113,A -85,B 0,C 180,E1 -27889.999,E2 -27889.999} C_VEL
LIN {X 0,Y 85.728,Z 1007.586,A -85,B 0,C 180,E1 -27894.71,E2 -27894.71} C_VEL
LIN {X 0,Y 85.668,Z 999.368,A -85,B 0,C 180,E1 -27897.651,E2 -27897.651} C_VEL
LIN {X 0,Y 85.7,Z 988.881,A -85,B 0,C 180,E1 -27900.59,E2 -27900.59} C_VEL
LIN {X 0,Y 85.531,Z 977.824,A -85,B 0,C 180,E1 -27902.946,E2 -27902.946} C_VEL
LIN {X 0,Y 84.667,Z 942.182,A -85,B 0,C 180,E1 -27909.709,E2 -27909.709} C_VEL
LIN {X 0,Y 84.473,Z 935.662,A -85,B 0,C 180,E1 -27910.867,E2 -27910.867} C_VEL
LIN {X 0,Y 82.242,Z 925.048,A -85,B 0,C 180,E1 -27912.338,E2 -27912.338} C_VEL
LIN {X 0,Y 79.561,Z 925.383,A -85,B 0,C 180,E1 -27927.953,E2 -27927.953} C_VEL
LIN {X 0,Y 79.331,Z 925.403,A -85,B 0,C 180,E1 -27933.597,E2 -27933.597} C_VEL
LIN {X 0,Y 78.577,Z 925.503,A -85,B 0,C 180,E1 -27937.838,E2 -27937.838} C_VEL
LIN {X 0,Y 76.977,Z 925.706,A -85,B 0,C 180,E1 -27942.057,E2 -27942.057} C_VEL
LIN {X 0,Y 72.499,Z 926.266,A -85,B 0,C 180,E1 -27954.043,E2 -27954.043} C_VEL
LIN {X 0,Y 72.203,Z 926.287,A -85,B 0,C 180,E1 -27957.264,E2 -27957.264} C_VEL
LIN {X 0,Y 72.36,Z 926.283,A -85,B 0,C 180,E1 -27960.948,E2 -27960.948} C_VEL
LIN {X 0,Y 72.371,Z 926.273,A -85,B 0,C 180,E1 -27967.143,E2 -27967.143} C_VEL
LIN {X 0,Y 72.682,Z 926.234,A -85,B 0,C 180,E1 -27975.241,E2 -27975.241} C_VEL
LIN {X 0,Y 72.83,Z 926.223,A -85,B 0,C 180,E1 -27978.873,E2 -27978.873} C_VEL
LIN {X 0,Y 73.534,Z 926.139,A -85,B 0,C 180,E1 -27990.001,E2 -27990.001} C_VEL
LIN {X 0,Y 72.83,Z 926.223,A -85,B 0,C 180,E1 -28001.129,E2 -28001.129} C_VEL
LIN {X 0,Y 72.506,Z 926.264,A -85,B 0,C 180,E1 -28006.906,E2 -28006.906} C_VEL
LIN {X 0,Y 72.364,Z 926.273,A -85,B 0,C 180,E1 -28012.861,E2 -28012.861} C_VEL
LIN {X 0,Y 72.361,Z 926.282,A -85,B 0,C 180,E1 -28019.054,E2 -28019.054} C_VEL
LIN {X 0,Y 72.292,Z 926.291,A -85,B 0,C 180,E1 -28025.684,E2 -28025.684} C_VEL
LIN {X 0,Y 72.248,Z 926.29,A -85,B 0,C 180,E1 -28032.918,E2 -28032.918} C_VEL
LIN {X 0,Y 72.294,Z 926.282,A -85,B 0,C 180,E1 -28041.053,E2 -28041.053} C_VEL
LIN {X 0,Y 72.292,Z 926.292,A -85,B 0,C 180,E1 -28044.314,E2 -28044.314} C_VEL
LIN {X 0,Y 72.361,Z 926.275,A -85,B 0,C 180,E1 -28050.944,E2 -28050.944} C_VEL
LIN {X 0,Y 72.368,Z 926.278,A -85,B 0,C 180,E1 -28057.138,E2 -28057.138} C_VEL
LIN {X 0,Y 72.68,Z 926.243,A -85,B 0,C 180,E1 -28065.24,E2 -28065.24} C_VEL
LIN {X 0,Y 72.812,Z 926.217,A -85,B 0,C 180,E1 -28068.867,E2 -28068.867} C_VEL
LIN {X 0,Y 73.53,Z 926.134,A -85,B 0,C 180,E1 -28079.997,E2 -28079.997} C_VEL
LIN {X 0,Y 72.81,Z 926.228,A -85,B 0,C 180,E1 -28091.128,E2 -28091.128} C_VEL
LIN {X 0,Y 72.503,Z 926.257,A -85,B 0,C 180,E1 -28096.903,E2 -28096.903} C_VEL
LIN {X 0,Y 72.36,Z 926.28,A -85,B 0,C 180,E1 -28102.858,E2 -28102.858} C_VEL
LIN {X 0,Y 72.358,Z 926.284,A -85,B 0,C 180,E1 -28109.052,E2 -28109.052} C_VEL
LIN {X 0,Y 72.288,Z 926.284,A -85,B 0,C 180,E1 -28115.682,E2 -28115.682} C_VEL
LIN {X 0,Y 72.241,Z 926.29,A -85,B 0,C 180,E1 -28122.918,E2 -28122.918} C_VEL
LIN {X 0,Y 72.304,Z 926.286,A -85,B 0,C 180,E1 -28131.038,E2 -28131.038} C_VEL
LIN {X 0,Y 72.746,Z 926.227,A -85,B 0,C 180,E1 -28141.114,E2 -28141.114} C_VEL
LIN {X 0,Y 72.978,Z 926.208,A -85,B 0,C 180,E1 -28147.342,E2 -28147.342} C_VEL
LIN {X 0,Y 74.878,Z 925.97,A -85,B 0,C 180,E1 -28158.837,E2 -28158.837} C_VEL
LIN {X 0,Y 77.185,Z 949.382,A -85,B 0,C 180,E1 -28163.07,E2 -28163.07} C_VEL
LIN {X 0,Y 79.683,Z 966.849,A -85,B 0,C 180,E1 -28165.89,E2 -28165.89} C_VEL
LIN {X 0,Y 81.102,Z 993.243,A -85,B 0,C 180,E1 -28171.396,E2 -28171.396} C_VEL
LIN {X 0,Y 81.743,Z 1003.958,A -85,B 0,C 180,E1 -28174.314,E2 -28174.314} C_VEL
LIN {X 0,Y 82.433,Z 1013.934,A -85,B 0,C 180,E1 -28177.963,E2 -28177.963} C_VEL
LIN {X 0,Y 83.224,Z 1021.447,A -85,B 0,C 180,E1 -28181.394,E2 -28181.394} C_VEL
LIN {X 0,Y 83.578,Z 1024.73,A -85,B 0,C 180,E1 -28183.253,E2 -28183.253} C_VEL
LIN {X 0,Y 83.594,Z 1028.179,A -85,B 0,C 180,E1 -28185.857,E2 -28185.857} C_VEL
LIN {X 0,Y 84.159,Z 1037.327,A -85,B 0,C 180,E1 -28194.679,E2 -28194.679} C_VEL
LIN {X 0,Y 86.686,Z 1043.764,A -85,B 0,C 180,E1 -28201.801,E2 -28201.801} C_VEL
LIN {X 0,Y 90.833,Z 1049.397,A -85,B 0,C 180,E1 -28208.241,E2 -28208.241} C_VEL
LIN {X 0,Y 98.397,Z 1055.557,A -85,B 0,C 180,E1 -28215.581,E2 -28215.581} C_VEL
LIN {X 0,Y 97.36,Z 1054.685,A -85,B 0,C 180,E1 -28216.704,E2 -28216.704} C_VEL
LIN {X 0,Y 89.359,Z 1046.295,A -85,B 0,C 180,E1 -28224.014,E2 -28224.014} C_VEL
LIN {X 0,Y 85.099,Z 1039.013,A -85,B 0,C 180,E1 -28230.298,E2 -28230.298} C_VEL
LIN {X 0,Y 82.169,Z 1030.286,A -85,B 0,C 180,E1 -28237.365,E2 -28237.365} C_VEL
LIN {X 0,Y 81.079,Z 1021.849,A -85,B 0,C 180,E1 -28243.51,E2 -28243.51} C_VEL
LIN {X 0,Y 80.637,Z 1015.335,A -85,B 0,C 180,E1 -28247.415,E2 -28247.415} C_VEL
LIN {X 0,Y 80.181,Z 1006.892,A -85,B 0,C 180,E1 -28251.496,E2 -28251.496} C_VEL
LIN {X 0,Y 79.933,Z 997.811,A -85,B 0,C 180,E1 -28254.958,E2 -28254.958} C_VEL
LIN {X 0,Y 79.832,Z 986.573,A -85,B 0,C 180,E1 -28258.229,E2 -28258.229} C_VEL
LIN {X 0,Y 79.502,Z 975.969,A -85,B 0,C 180,E1 -28260.556,E2 -28260.556} C_VEL
LIN {X 0,Y 78.154,Z 937.858,A -85,B 0,C 180,E1 -28268.441,E2 -28268.441} C_VEL
LIN {X 0,Y 77.442,Z 933.302,A -85,B 0,C 180,E1 -28269.141,E2 -28269.141} C_VEL
LIN {X 0,Y 75.814,Z 925.849,A -85,B 0,C 180,E1 -28270.273,E2 -28270.273} C_VEL
LIN {X 0,Y 72.445,Z 926.264,A -85,B 0,C 180,E1 -28289.18,E2 -28289.18} C_VEL
LIN {X 0,Y 72.293,Z 926.282,A -85,B 0,C 180,E1 -28298.948,E2 -28298.948} C_VEL
LIN {X 0,Y 72.246,Z 926.291,A -85,B 0,C 180,E1 -28307.083,E2 -28307.083} C_VEL
LIN {X 0,Y 72.293,Z 926.291,A -85,B 0,C 180,E1 -28314.318,E2 -28314.318} C_VEL
LIN {X 0,Y 72.203,Z 926.287,A -85,B 0,C 180,E1 -28317.264,E2 -28317.264} C_VEL
LIN {X 0,Y 71.892,Z 926.339,A -85,B 0,C 180,E1 -28320.376,E2 -28320.376} C_VEL
LIN {X 0,Y 70.574,Z 926.508,A -85,B 0,C 180,E1 -28325.02,E2 -28325.02} C_VEL
LIN {X 0,Y 67.552,Z 926.881,A -85,B 0,C 180,E1 -28332.993,E2 -28332.993} C_VEL
LIN {X 0,Y 65.908,Z 927.087,A -85,B 0,C 180,E1 -28339.884,E2 -28339.884} C_VEL
LIN {X 0,Y 65.847,Z 927.084,A -85,B 0,C 180,E1 -28343.437,E2 -28343.437} C_VEL
LIN {X 0,Y 66.434,Z 927.023,A -85,B 0,C 180,E1 -28350.001,E2 -28350.001} C_VEL
LIN {X 0,Y 65.724,Z 927.103,A -85,B 0,C 180,E1 -28362.35,E2 -28362.35} C_VEL
LIN {X 0,Y 65.337,Z 927.159,A -85,B 0,C 180,E1 -28368.827,E2 -28368.827} C_VEL
LIN {X 0,Y 65.216,Z 927.17,A -85,B 0,C 180,E1 -28375.536,E2 -28375.536} C_VEL
LIN {X 0,Y 65.171,Z 927.169,A -85,B 0,C 180,E1 -28382.63,E2 -28382.63} C_VEL
LIN {X 0,Y 65.182,Z 927.168,A -85,B 0,C 180,E1 -28390.992,E2 -28390.992} C_VEL
LIN {X 0,Y 65.202,Z 927.166,A -85,B 0,C 180,E1 -28399.701,E2 -28399.701} C_VEL
LIN {X 0,Y 65.227,Z 927.162,A -85,B 0,C 180,E1 -28409.542,E2 -28409.542} C_VEL
LIN {X 0,Y 65.218,Z 927.174,A -85,B 0,C 180,E1 -28414.463,E2 -28414.463} C_VEL
LIN {X 0,Y 65.582,Z 927.128,A -85,B 0,C 180,E1 -28424.685,E2 -28424.685} C_VEL
LIN {X 0,Y 65.692,Z 927.104,A -85,B 0,C 180,E1 -28427.642,E2 -28427.642} C_VEL
LIN {X 0,Y 66.429,Z 927.018,A -85,B 0,C 180,E1 -28439.997,E2 -28439.997} C_VEL
LIN {X 0,Y 65.711,Z 927.112,A -85,B 0,C 180,E1 -28452.348,E2 -28452.348} C_VEL
LIN {X 0,Y 65.333,Z 927.156,A -85,B 0,C 180,E1 -28458.824,E2 -28458.824} C_VEL
LIN {X 0,Y 65.211,Z 927.164,A -85,B 0,C 180,E1 -28465.534,E2 -28465.534} C_VEL
LIN {X 0,Y 65.167,Z 927.174,A -85,B 0,C 180,E1 -28472.628,E2 -28472.628} C_VEL
LIN {X 0,Y 65.177,Z 927.176,A -85,B 0,C 180,E1 -28480.99,E2 -28480.99} C_VEL
LIN {X 0,Y 65.207,Z 927.174,A -85,B 0,C 180,E1 -28489.707,E2 -28489.707} C_VEL
LIN {X 0,Y 65.505,Z 927.136,A -85,B 0,C 180,E1 -28499.123,E2 -28499.123} C_VEL
LIN {X 0,Y 65.743,Z 927.104,A -85,B 0,C 180,E1 -28504.683,E2 -28504.683} C_VEL
LIN {X 0,Y 68.553,Z 926.756,A -85,B 0,C 180,E1 -28521.524,E2 -28521.524} C_VEL
LIN {X 0,Y 71.302,Z 950.33,A -85,B 0,C 180,E1 -28526.113,E2 -28526.113} C_VEL
LIN {X 0,Y 73.821,Z 967.052,A -85,B 0,C 180,E1 -28528.976,E2 -28528.976} C_VEL
LIN {X 0,Y 75.563,Z 992.009,A -85,B 0,C 180,E1 -28534.5,E2 -28534.5} C_VEL
LIN {X 0,Y 76.306,Z 1001.839,A -85,B 0,C 180,E1 -28537.275,E2 -28537.275} C_VEL
LIN {X 0,Y 77.137,Z 1010.43,A -85,B 0,C 180,E1 -28540.498,E2 -28540.498} C_VEL
LIN {X 0,Y 78.221,Z 1018.543,A -85,B 0,C 180,E1 -28544.304,E2 -28544.304} C_VEL
LIN {X 0,Y 78.674,Z 1023.178,A -85,B 0,C 180,E1 -28547.193,E2 -28547.193} C_VEL
LIN {X 0,Y 79.001,Z 1030.852,A -85,B 0,C 180,E1 -28554.518,E2 -28554.518} C_VEL
LIN {X 0,Y 81.926,Z 1039.345,A -85,B 0,C 180,E1 -28563.889,E2 -28563.889} C_VEL
LIN {X 0,Y 86.324,Z 1045.306,A -85,B 0,C 180,E1 -28570.64,E2 -28570.64} C_VEL
LIN {X 0,Y 89.952,Z 1048.806,A -85,B 0,C 180,E1 -28574.681,E2 -28574.681} C_VEL
LIN {X 0,Y 90.562,Z 1049.267,A -85,B 0,C 180,E1 -28575.701,E2 -28575.701} C_VEL
LIN {X 0,Y 82.98,Z 1040.023,A -85,B 0,C 180,E1 -28583.642,E2 -28583.642} C_VEL
LIN {X 0,Y 78.856,Z 1031.638,A -85,B 0,C 180,E1 -28590.65,E2 -28590.65} C_VEL
LIN {X 0,Y 76.46,Z 1021.796,A -85,B 0,C 180,E1 -28598.431,E2 -28598.431} C_VEL
LIN {X 0,Y 75.716,Z 1014.824,A -85,B 0,C 180,E1 -28603.133,E2 -28603.133} C_VEL
LIN {X 0,Y 74.964,Z 1004.846,A -85,B 0,C 180,E1 -28608.293,E2 -28608.293} C_VEL
LIN {X 0,Y 74.519,Z 995.921,A -85,B 0,C 180,E1 -28611.87,E2 -28611.87} C_VEL
LIN {X 0,Y 74.202,Z 983.628,A -85,B 0,C 180,E1 -28615.589,E2 -28615.589} C_VEL
LIN {X 0,Y 72.783,Z 957.48,A -85,B 0,C 180,E1 -28621.559,E2 -28621.559} C_VEL
LIN {X 0,Y 71.712,Z 935.809,A -85,B 0,C 180,E1 -28626.285,E2 -28626.285} C_VEL
LIN {X 0,Y 69.594,Z 926.63,A -85,B 0,C 180,E1 -28627.653,E2 -28627.653} C_VEL
LIN {X 0,Y 65.49,Z 927.14,A -85,B 0,C 180,E1 -28645.424,E2 -28645.424} C_VEL
LIN {X 0,Y 65.224,Z 927.17,A -85,B 0,C 180,E1 -28652.603,E2 -28652.603} C_VEL
LIN {X 0,Y 65.181,Z 927.171,A -85,B 0,C 180,E1 -28660.997,E2 -28660.997} C_VEL
LIN {X 0,Y 65.201,Z 927.167,A -85,B 0,C 180,E1 -28669.705,E2 -28669.705} C_VEL
LIN {X 0,Y 65.226,Z 927.166,A -85,B 0,C 180,E1 -28679.546,E2 -28679.546} C_VEL
LIN {X 0,Y 65.219,Z 927.169,A -85,B 0,C 180,E1 -28684.468,E2 -28684.468} C_VEL
LIN {X 0,Y 65.584,Z 927.12,A -85,B 0,C 180,E1 -28694.687,E2 -28694.687} C_VEL
LIN {X 0,Y 65.724,Z 927.103,A -85,B 0,C 180,E1 -28697.652,E2 -28697.652} C_VEL
LIN {X 0,Y 65.847,Z 927.084,A -85,B 0,C 180,E1 -28703.437,E2 -28703.437} C_VEL
LIN {X 0,Y 65.714,Z 927.12,A -85,B 0,C 180,E1 -28706.836,E2 -28706.836} C_VEL
LIN {X 0,Y 64.431,Z 927.299,A -85,B 0,C 180,E1 -28711.911,E2 -28711.911} C_VEL
LIN {X 0,Y 62.46,Z 927.55,A -85,B 0,C 180,E1 -28717.006,E2 -28717.006} C_VEL
LIN {X 0,Y 58.088,Z 928.047,A -85,B 0,C 180,E1 -28732.395,E2 -28732.395} C_VEL
LIN {X 0,Y 58.136,Z 928.045,A -85,B 0,C 180,E1 -28742.19,E2 -28742.19} C_VEL
LIN {X 0,Y 58.024,Z 928.07,A -85,B 0,C 180,E1 -28747.275,E2 -28747.275} C_VEL
LIN {X 0,Y 58.012,Z 928.071,A -85,B 0,C 180,E1 -28756.628,E2 -28756.628} C_VEL
LIN {X 0,Y 58.024,Z 928.063,A -85,B 0,C 180,E1 -28762.723,E2 -28762.723} C_VEL
LIN {X 0,Y 58.127,Z 928.047,A -85,B 0,C 180,E1 -28771.074,E2 -28771.074} C_VEL
LIN {X 0,Y 58.159,Z 928.042,A -85,B 0,C 180,E1 -28778.741,E2 -28778.741} C_VEL
LIN {X 0,Y 58.565,Z 927.997,A -85,B 0,C 180,E1 -28786.11,E2 -28786.11} C_VEL
LIN {X 0,Y 58.756,Z 927.979,A -85,B 0,C 180,E1 -28793.127,E2 -28793.127} C_VEL
LIN {X 0,Y 59.322,Z 927.903,A -85,B 0,C 180,E1 -28799.997,E2 -28799.997} C_VEL
LIN {X 0,Y 58.756,Z 927.968,A -85,B 0,C 180,E1 -28806.867,E2 -28806.867} C_VEL
LIN {X 0,Y 58.455,Z 928.005,A -85,B 0,C 180,E1 -28815.875,E2 -28815.875} C_VEL
LIN {X 0,Y 58.154,Z 928.053,A -85,B 0,C 180,E1 -28821.254,E2 -28821.254} C_VEL
LIN {X 0,Y 58.123,Z 928.056,A -85,B 0,C 180,E1 -28828.921,E2 -28828.921} C_VEL
LIN {X 0,Y 58.019,Z 928.067,A -85,B 0,C 180,E1 -28837.273,E2 -28837.273} C_VEL
LIN {X 0,Y 58.013,Z 928.068,A -85,B 0,C 180,E1 -28846.62,E2 -28846.62} C_VEL
LIN {X 0,Y 58.332,Z 928.032,A -85,B 0,C 180,E1 -28857.493,E2 -28857.493} C_VEL
LIN {X 0,Y 58.476,Z 928.004,A -85,B 0,C 180,E1 -28861.265,E2 -28861.265} C_VEL
LIN {X 0,Y 59.172,Z 927.919,A -85,B 0,C 180,E1 -28871.828,E2 -28871.828} C_VEL
LIN {X 0,Y 62.559,Z 927.505,A -85,B 0,C 180,E1 -28884.953,E2 -28884.953} C_VEL
LIN {X 0,Y 65.674,Z 951.327,A -85,B 0,C 180,E1 -28889.698,E2 -28889.698} C_VEL
LIN {X 0,Y 68.159,Z 966.47,A -85,B 0,C 180,E1 -28892.4,E2 -28892.4} C_VEL
LIN {X 0,Y 70.367,Z 990.321,A -85,B 0,C 180,E1 -28898.073,E2 -28898.073} C_VEL
LIN {X 0,Y 71.453,Z 1001.162,A -85,B 0,C 180,E1 -28901.344,E2 -28901.344} C_VEL
LIN {X 0,Y 72.492,Z 1009.579,A -85,B 0,C 180,E1 -28904.742,E2 -28904.742} C_VEL
LIN {X 0,Y 73.609,Z 1016.421,A -85,B 0,C 180,E1 -28908.076,E2 -28908.076} C_VEL
LIN {X 0,Y 73.932,Z 1018.597,A -85,B 0,C 180,E1 -28909.433,E2 -28909.433} C_VEL
LIN {X 0,Y 74.31,Z 1024.7,A -85,B 0,C 180,E1 -28915.19,E2 -28915.19} C_VEL
LIN {X 0,Y 76.676,Z 1033.135,A -85,B 0,C 180,E1 -28924.423,E2 -28924.423} C_VEL
LIN {X 0,Y 82.087,Z 1041.016,A -85,B 0,C 180,E1 -28933.229,E2 -28933.229} C_VEL
LIN {X 0,Y 83.038,Z 1041.972,A -85,B 0,C 180,E1 -28935.709,E2 -28935.709} C_VEL
LIN {X 0,Y 76.781,Z 1032.713,A -85,B 0,C 180,E1 -28943.493,E2 -28943.493} C_VEL
LIN {X 0,Y 73.47,Z 1024.921,A -85,B 0,C 180,E1 -28949.942,E2 -28949.942} C_VEL
LIN {X 0,Y 71.733,Z 1016.969,A -85,B 0,C 180,E1 -28956.164,E2 -28956.164} C_VEL
LIN {X 0,Y 70.723,Z 1009.374,A -85,B 0,C 180,E1 -28961.144,E2 -28961.144} C_VEL
LIN {X 0,Y 69.908,Z 1000.815,A -85,B 0,C 180,E1 -28965.446,E2 -28965.446} C_VEL
LIN {X 0,Y 69.351,Z 991.05,A -85,B 0,C 180,E1 -28969.234,E2 -28969.234} C_VEL
LIN {X 0,Y 68.706,Z 978.116,A -85,B 0,C 180,E1 -28973.026,E2 -28973.026} C_VEL
LIN {X 0,Y 65.718,Z 936.726,A -85,B 0,C 180,E1 -28983.068,E2 -28983.068} C_VEL
LIN {X 0,Y 63.559,Z 927.379,A -85,B 0,C 180,E1 -28984.527,E2 -28984.527} C_VEL
LIN {X 0,Y 60.065,Z 927.811,A -85,B 0,C 180,E1 -28993.537,E2 -28993.537} C_VEL
LIN {X 0,Y 58.259,Z 928.031,A -85,B 0,C 180,E1 -29008.855,E2 -29008.855} C_VEL
LIN {X 0,Y 58.039,Z 928.061,A -85,B 0,C 180,E1 -29017.266,E2 -29017.266} C_VEL
LIN {X 0,Y 58.01,Z 928.064,A -85,B 0,C 180,E1 -29026.632,E2 -29026.632} C_VEL
LIN {X 0,Y 58.023,Z 928.07,A -85,B 0,C 180,E1 -29032.728,E2 -29032.728} C_VEL
LIN {X 0,Y 58.128,Z 928.055,A -85,B 0,C 180,E1 -29041.079,E2 -29041.079} C_VEL
LIN {X 0,Y 58.161,Z 928.046,A -85,B 0,C 180,E1 -29048.747,E2 -29048.747} C_VEL
LIN {X 0,Y 58.596,Z 927.987,A -85,B 0,C 180,E1 -29056.122,E2 -29056.122} C_VEL
LIN {X 0,Y 58.782,Z 927.967,A -85,B 0,C 180,E1 -29063.609,E2 -29063.609} C_VEL
LIN {X 0,Y 59.328,Z 927.908,A -85,B 0,C 180,E1 -29070.001,E2 -29070.001} C_VEL
LIN {X 0,Y 58.77,Z 927.971,A -85,B 0,C 180,E1 -29076.869,E2 -29076.869} C_VEL
LIN {X 0,Y 58.458,Z 928.009,A -85,B 0,C 180,E1 -29085.879,E2 -29085.879} C_VEL
LIN {X 0,Y 58.088,Z 928.047,A -85,B 0,C 180,E1 -29092.395,E2 -29092.395} C_VEL
LIN {X 0,Y 57.58,Z 928.123,A -85,B 0,C 180,E1 -29096.254,E2 -29096.254} C_VEL
LIN {X 0,Y 56.019,Z 928.318,A -85,B 0,C 180,E1 -29102.021,E2 -29102.021} C_VEL
LIN {X 0,Y 52.728,Z 928.73,A -85,B 0,C 180,E1 -29112.091,E2 -29112.091} C_VEL
LIN {X 0,Y 51.025,Z 928.93,A -85,B 0,C 180,E1 -29120.997,E2 -29120.997} C_VEL
LIN {X 0,Y 51.002,Z 928.943,A -85,B 0,C 180,E1 -29125.613,E2 -29125.613} C_VEL
LIN {X 0,Y 51,Z 928.944,A -85,B 0,C 180,E1 -29135.577,E2 -29135.577} C_VEL
LIN {X 0,Y 51.395,Z 928.896,A -85,B 0,C 180,E1 -29144.124,E2 -29144.124} C_VEL
LIN {X 0,Y 51.63,Z 928.865,A -85,B 0,C 180,E1 -29152.173,E2 -29152.173} C_VEL
LIN {X 0,Y 52.207,Z 928.788,A -85,B 0,C 180,E1 -29159.996,E2 -29159.996} C_VEL
LIN {X 0,Y 51.635,Z 928.855,A -85,B 0,C 180,E1 -29167.819,E2 -29167.819} C_VEL
LIN {X 0,Y 51.336,Z 928.892,A -85,B 0,C 180,E1 -29176.598,E2 -29176.598} C_VEL
LIN {X 0,Y 50.996,Z 928.935,A -85,B 0,C 180,E1 -29184.418,E2 -29184.418} C_VEL
LIN {X 0,Y 50.984,Z 928.935,A -85,B 0,C 180,E1 -29194.197,E2 -29194.197} C_VEL
LIN {X 0,Y 50.977,Z 928.936,A -85,B 0,C 180,E1 -29203.572,E2 -29203.572} C_VEL
LIN {X 0,Y 51.219,Z 928.916,A -85,B 0,C 180,E1 -29216.71,E2 -29216.71} C_VEL
LIN {X 0,Y 51.546,Z 928.877,A -85,B 0,C 180,E1 -29225.854,E2 -29225.854} C_VEL
LIN {X 0,Y 56.254,Z 928.286,A -85,B 0,C 180,E1 -29248.037,E2 -29248.037} C_VEL
LIN {X 0,Y 56.932,Z 928.421,A -85,B 0,C 180,E1 -29249.174,E2 -29249.174} C_VEL
LIN {X 0,Y 60.459,Z 951.866,A -85,B 0,C 180,E1 -29254.061,E2 -29254.061} C_VEL
LIN {X 0,Y 62.998,Z 965.952,A -85,B 0,C 180,E1 -29256.625,E2 -29256.625} C_VEL
LIN {X 0,Y 65.691,Z 989.616,A -85,B 0,C 180,E1 -29262.55,E2 -29262.55} C_VEL
LIN {X 0,Y 67.032,Z 1000.434,A -85,B 0,C 180,E1 -29265.974,E2 -29265.974} C_VEL
LIN {X 0,Y 68.341,Z 1008.749,A -85,B 0,C 180,E1 -29269.524,E2 -29269.524} C_VEL
LIN {X 0,Y 69.422,Z 1014.124,A -85,B 0,C 180,E1 -29272.31,E2 -29272.31} C_VEL
LIN {X 0,Y 69.788,Z 1017.195,A -85,B 0,C 180,E1 -29275.001,E2 -29275.001} C_VEL
LIN {X 0,Y 71.306,Z 1025.04,A -85,B 0,C 180,E1 -29283.313,E2 -29283.313} C_VEL
LIN {X 0,Y 76.232,Z 1033.981,A -85,B 0,C 180,E1 -29293.379,E2 -29293.379} C_VEL
LIN {X 0,Y 77.088,Z 1035.096,A -85,B 0,C 180,E1 -29294.772,E2 -29294.772} C_VEL
LIN {X 0,Y 71.722,Z 1026.241,A -85,B 0,C 180,E1 -29302.058,E2 -29302.058} C_VEL
LIN {X 0,Y 68.18,Z 1016.219,A -85,B 0,C 180,E1 -29310.343,E2 -29310.343} C_VEL
LIN {X 0,Y 66.766,Z 1008.345,A -85,B 0,C 180,E1 -29315.93,E2 -29315.93} C_VEL
LIN {X 0,Y 65.655,Z 1000.073,A -85,B 0,C 180,E1 -29320.46,E2 -29320.46} C_VEL
LIN {X 0,Y 64.834,Z 991.668,A -85,B 0,C 180,E1 -29324.077,E2 -29324.077} C_VEL
LIN {X 0,Y 63.889,Z 979.348,A -85,B 0,C 180,E1 -29328.1,E2 -29328.1} C_VEL
LIN {X 0,Y 60.764,Z 947.077,A -85,B 0,C 180,E1 -29336.48,E2 -29336.48} C_VEL
LIN {X 0,Y 59.751,Z 935.548,A -85,B 0,C 180,E1 -29339.395,E2 -29339.395} C_VEL
LIN {X 0,Y 57.888,Z 928.082,A -85,B 0,C 180,E1 -29340.583,E2 -29340.583} C_VEL
LIN {X 0,Y 54.586,Z 928.499,A -85,B 0,C 180,E1 -29347.401,E2 -29347.401} C_VEL
LIN {X 0,Y 51.364,Z 928.898,A -85,B 0,C 180,E1 -29364.239,E2 -29364.239} C_VEL
LIN {X 0,Y 51.05,Z 928.939,A -85,B 0,C 180,E1 -29374.311,E2 -29374.311} C_VEL
LIN {X 0,Y 50.977,Z 928.94,A -85,B 0,C 180,E1 -29386.425,E2 -29386.425} C_VEL
LIN {X 0,Y 51.014,Z 928.933,A -85,B 0,C 180,E1 -29396.561,E2 -29396.561} C_VEL
LIN {X 0,Y 51.001,Z 928.935,A -85,B 0,C 180,E1 -29405.583,E2 -29405.583} C_VEL
LIN {X 0,Y 51.395,Z 928.888,A -85,B 0,C 180,E1 -29414.13,E2 -29414.13} C_VEL
LIN {X 0,Y 51.648,Z 928.862,A -85,B 0,C 180,E1 -29422.181,E2 -29422.181} C_VEL
LIN {X 0,Y 52.216,Z 928.794,A -85,B 0,C 180,E1 -29430.001,E2 -29430.001} C_VEL
LIN {X 0,Y 51.647,Z 928.862,A -85,B 0,C 180,E1 -29437.822,E2 -29437.822} C_VEL
LIN {X 0,Y 51.34,Z 928.898,A -85,B 0,C 180,E1 -29446.602,E2 -29446.602} C_VEL
LIN {X 0,Y 51,Z 928.935,A -85,B 0,C 180,E1 -29454.421,E2 -29454.421} C_VEL
LIN {X 0,Y 50.988,Z 928.938,A -85,B 0,C 180,E1 -29464.2,E2 -29464.2} C_VEL
LIN {X 0,Y 50.979,Z 928.94,A -85,B 0,C 180,E1 -29473.577,E2 -29473.577} C_VEL
LIN {X 0,Y 51.002,Z 928.943,A -85,B 0,C 180,E1 -29485.613,E2 -29485.613} C_VEL
LIN {X 0,Y 50.675,Z 929.004,A -85,B 0,C 180,E1 -29489.214,E2 -29489.214} C_VEL
LIN {X 0,Y 48.957,Z 929.218,A -85,B 0,C 180,E1 -29494.129,E2 -29494.129} C_VEL
LIN {X 0,Y 44.514,Z 929.744,A -85,B 0,C 180,E1 -29506.596,E2 -29506.596} C_VEL
LIN {X 0,Y 44.416,Z 929.754,A -85,B 0,C 180,E1 -29510.16,E2 -29510.16} C_VEL
LIN {X 0,Y 45.083,Z 929.675,A -85,B 0,C 180,E1 -29519.996,E2 -29519.996} C_VEL
LIN {X 0,Y 44.48,Z 929.749,A -85,B 0,C 180,E1 -29529.087,E2 -29529.087} C_VEL
LIN {X 0,Y 44.105,Z 929.797,A -85,B 0,C 180,E1 -29538.58,E2 -29538.58} C_VEL
LIN {X 0,Y 43.811,Z 929.838,A -85,B 0,C 180,E1 -29548.762,E2 -29548.762} C_VEL
LIN {X 0,Y 43.785,Z 929.843,A -85,B 0,C 180,E1 -29559.94,E2 -29559.94} C_VEL
LIN {X 0,Y 43.953,Z 929.811,A -85,B 0,C 180,E1 -29573.075,E2 -29573.075} C_VEL
LIN {X 0,Y 44.199,Z 929.781,A -85,B 0,C 180,E1 -29581.507,E2 -29581.507} C_VEL
LIN {X 0,Y 44.976,Z 929.685,A -85,B 0,C 180,E1 -29591.787,E2 -29591.787} C_VEL
LIN {X 0,Y 49.302,Z 929.148,A -85,B 0,C 180,E1 -29609.998,E2 -29609.998} C_VEL
LIN {X 0,Y 51.617,Z 928.866,A -85,B 0,C 180,E1 -29614.147,E2 -29614.147} C_VEL
LIN {X 0,Y 55.361,Z 950.881,A -85,B 0,C 180,E1 -29618.948,E2 -29618.948} C_VEL
LIN {X 0,Y 58.267,Z 965.651,A -85,B 0,C 180,E1 -29621.637,E2 -29621.637} C_VEL
LIN {X 0,Y 61.519,Z 988.699,A -85,B 0,C 180,E1 -29627.664,E2 -29627.664} C_VEL
LIN {X 0,Y 63.194,Z 999.353,A -85,B 0,C 180,E1 -29631.187,E2 -29631.187} C_VEL
LIN {X 0,Y 65.199,Z 1008.885,A -85,B 0,C 180,E1 -29635.541,E2 -29635.541} C_VEL
LIN {X 0,Y 65.736,Z 1011.32,A -85,B 0,C 180,E1 -29637.024,E2 -29637.024} C_VEL
LIN {X 0,Y 66.572,Z 1016.609,A -85,B 0,C 180,E1 -29642.38,E2 -29642.38} C_VEL
LIN {X 0,Y 70.345,Z 1025.549,A -85,B 0,C 180,E1 -29652.545,E2 -29652.545} C_VEL
LIN {X 0,Y 71.061,Z 1026.732,A -85,B 0,C 180,E1 -29653.812,E2 -29653.812} C_VEL
LIN {X 0,Y 70.224,Z 1025.369,A -85,B 0,C 180,E1 -29655.532,E2 -29655.532} C_VEL
LIN {X 0,Y 65.673,Z 1015.572,A -85,B 0,C 180,E1 -29663.515,E2 -29663.515} C_VEL
LIN {X 0,Y 63.643,Z 1008.277,A -85,B 0,C 180,E1 -29669.291,E2 -29669.291} C_VEL
LIN {X 0,Y 62.422,Z 1002.082,A -85,B 0,C 180,E1 -29673.237,E2 -29673.237} C_VEL
LIN {X 0,Y 61.15,Z 992.768,A -85,B 0,C 180,E1 -29677.846,E2 -29677.846} C_VEL
LIN {X 0,Y 59.777,Z 980.002,A -85,B 0,C 180,E1 -29682.469,E2 -29682.469} C_VEL
LIN {X 0,Y 55.854,Z 948.8,A -85,B 0,C 180,E1 -29691.181,E2 -29691.181} C_VEL
LIN {X 0,Y 54.412,Z 935.848,A -85,B 0,C 180,E1 -29694.676,E2 -29694.676} C_VEL
LIN {X 0,Y 52.622,Z 928.739,A -85,B 0,C 180,E1 -29695.663,E2 -29695.663} C_VEL
LIN {X 0,Y 49.212,Z 929.159,A -85,B 0,C 180,E1 -29701.53,E2 -29701.53} C_VEL
LIN {X 0,Y 44.719,Z 929.717,A -85,B 0,C 180,E1 -29719.45,E2 -29719.45} C_VEL
LIN {X 0,Y 44.03,Z 929.803,A -85,B 0,C 180,E1 -29728.615,E2 -29728.615} C_VEL
LIN {X 0,Y 43.807,Z 929.829,A -85,B 0,C 180,E1 -29739.926,E2 -29739.926} C_VEL
LIN {X 0,Y 43.815,Z 929.84,A -85,B 0,C 180,E1 -29753.331,E2 -29753.331} C_VEL
LIN {X 0,Y 43.815,Z 929.838,A -85,B 0,C 180,E1 -29761.238,E2 -29761.238} C_VEL
LIN {X 0,Y 44.183,Z 929.792,A -85,B 0,C 180,E1 -29772.645,E2 -29772.645} C_VEL
LIN {X 0,Y 44.495,Z 929.755,A -85,B 0,C 180,E1 -29780.914,E2 -29780.914} C_VEL
LIN {X 0,Y 45.093,Z 929.681,A -85,B 0,C 180,E1 -29790.002,E2 -29790.002} C_VEL
LIN {X 0,Y 44.49,Z 929.756,A -85,B 0,C 180,E1 -29799.091,E2 -29799.091} C_VEL
LIN {X 0,Y 44.108,Z 929.804,A -85,B 0,C 180,E1 -29808.585,E2 -29808.585} C_VEL
LIN {X 0,Y 43.815,Z 929.838,A -85,B 0,C 180,E1 -29818.766,E2 -29818.766} C_VEL
LIN {X 0,Y 43.788,Z 929.834,A -85,B 0,C 180,E1 -29829.944,E2 -29829.944} C_VEL
LIN {X 0,Y 43.831,Z 929.831,A -85,B 0,C 180,E1 -29843.297,E2 -29843.297} C_VEL
LIN {X 0,Y 43.815,Z 929.829,A -85,B 0,C 180,E1 -29851.231,E2 -29851.231} C_VEL
LIN {X 0,Y 44.182,Z 929.792,A -85,B 0,C 180,E1 -29862.642,E2 -29862.642} C_VEL
LIN {X 0,Y 44.416,Z 929.754,A -85,B 0,C 180,E1 -29870.16,E2 -29870.16} C_VEL
LIN {X 0,Y 44.179,Z 929.8,A -85,B 0,C 180,E1 -29874.284,E2 -29874.284} C_VEL
LIN {X 0,Y 42.595,Z 930.011,A -85,B 0,C 180,E1 -29879.953,E2 -29879.953} C_VEL
LIN {X 0,Y 37.006,Z 930.679,A -85,B 0,C 180,E1 -29898.644,E2 -29898.644} C_VEL
LIN {X 0,Y 36.694,Z 930.715,A -85,B 0,C 180,E1 -29915.065,E2 -29915.065} C_VEL
LIN {X 0,Y 36.715,Z 930.722,A -85,B 0,C 180,E1 -29920.029,E2 -29920.029} C_VEL
LIN {X 0,Y 36.779,Z 930.711,A -85,B 0,C 180,E1 -29929.842,E2 -29929.842} C_VEL
LIN {X 0,Y 36.882,Z 930.694,A -85,B 0,C 180,E1 -29935.131,E2 -29935.131} C_VEL
LIN {X 0,Y 37.572,Z 930.61,A -85,B 0,C 180,E1 -29949.259,E2 -29949.259} C_VEL
LIN {X 0,Y 42.188,Z 930.035,A -85,B 0,C 180,E1 -29971.894,E2 -29971.894} C_VEL
LIN {X 0,Y 47.01,Z 929.435,A -85,B 0,C 180,E1 -29980.514,E2 -29980.514} C_VEL
LIN {X 0,Y 51.332,Z 951.735,A -85,B 0,C 180,E1 -29985.218,E2 -29985.218} C_VEL
LIN {X 0,Y 54.135,Z 964.713,A -85,B 0,C 180,E1 -29987.469,E2 -29987.469} C_VEL
LIN {X 0,Y 58.007,Z 987.262,A -85,B 0,C 180,E1 -29993.414,E2 -29993.414} C_VEL
LIN {X 0,Y 60.048,Z 998.352,A -85,B 0,C 180,E1 -29997.125,E2 -29997.125} C_VEL
LIN {X 0,Y 61.949,Z 1006.212,A -85,B 0,C 180,E1 -30000.697,E2 -30000.697} C_VEL
LIN {X 0,Y 62.487,Z 1008.358,A -85,B 0,C 180,E1 -30002.291,E2 -30002.291} C_VEL
LIN {X 0,Y 64.832,Z 1015.892,A -85,B 0,C 180,E1 -30010.643,E2 -30010.643} C_VEL
LIN {X 0,Y 65.446,Z 1017.207,A -85,B 0,C 180,E1 -30012.158,E2 -30012.158} C_VEL
LIN {X 0,Y 65.734,Z 1017.834,A -85,B 0,C 180,E1 -30013.869,E2 -30013.869} C_VEL
LIN {X 0,Y 62.044,Z 1009.412,A -85,B 0,C 180,E1 -30020.738,E2 -30020.738} C_VEL
LIN {X 0,Y 59.979,Z 1002.046,A -85,B 0,C 180,E1 -30026.184,E2 -30026.184} C_VEL
LIN {X 0,Y 58.273,Z 993.897,A -85,B 0,C 180,E1 -30030.666,E2 -30030.666} C_VEL
LIN {X 0,Y 56.927,Z 985.028,A -85,B 0,C 180,E1 -30034.414,E2 -30034.414} C_VEL
LIN {X 0,Y 55.301,Z 973.819,A -85,B 0,C 180,E1 -30038.083,E2 -30038.083} C_VEL
LIN {X 0,Y 50.059,Z 938.652,A -85,B 0,C 180,E1 -30048.1,E2 -30048.1} C_VEL
LIN {X 0,Y 49.43,Z 935.066,A -85,B 0,C 180,E1 -30048.921,E2 -30048.921} C_VEL
LIN {X 0,Y 47.855,Z 929.334,A -85,B 0,C 180,E1 -30049.691,E2 -30049.691} C_VEL
LIN {X 0,Y 41.955,Z 930.065,A -85,B 0,C 180,E1 -30060.004,E2 -30060.004} C_VEL
LIN {X 0,Y 37.302,Z 930.64,A -85,B 0,C 180,E1 -30082.142,E2 -30082.142} C_VEL
LIN {X 0,Y 36.774,Z 930.717,A -85,B 0,C 180,E1 -30094.99,E2 -30094.99} C_VEL
LIN {X 0,Y 36.726,Z 930.711,A -85,B 0,C 180,E1 -30100.056,E2 -30100.056} C_VEL
LIN {X 0,Y 36.712,Z 930.714,A -85,B 0,C 180,E1 -30109.982,E2 -30109.982} C_VEL
LIN {X 0,Y 36.697,Z 930.72,A -85,B 0,C 180,E1 -30114.935,E2 -30114.935} C_VEL
LIN {X 0,Y 37.031,Z 930.685,A -85,B 0,C 180,E1 -30131.628,E2 -30131.628} C_VEL
LIN {X 0,Y 37.276,Z 930.649,A -85,B 0,C 180,E1 -30139.134,E2 -30139.134} C_VEL
LIN {X 0,Y 37.952,Z 930.57,A -85,B 0,C 180,E1 -30150.002,E2 -30150.002} C_VEL
LIN {X 0,Y 37.273,Z 930.649,A -85,B 0,C 180,E1 -30160.871,E2 -30160.871} C_VEL
LIN {X 0,Y 37.031,Z 930.685,A -85,B 0,C 180,E1 -30168.374,E2 -30168.374} C_VEL
LIN {X 0,Y 36.698,Z 930.72,A -85,B 0,C 180,E1 -30185.069,E2 -30185.069} C_VEL
LIN {X 0,Y 36.712,Z 930.714,A -85,B 0,C 180,E1 -30190.019,E2 -30190.019} C_VEL
LIN {X 0,Y 36.718,Z 930.712,A -85,B 0,C 180,E1 -30199.966,E2 -30199.966} C_VEL
LIN {X 0,Y 36.71,Z 930.725,A -85,B 0,C 180,E1 -30204.94,E2 -30204.94} C_VEL
LIN {X 0,Y 37.03,Z 930.677,A -85,B 0,C 180,E1 -30221.622,E2 -30221.622} C_VEL
LIN {X 0,Y 37.275,Z 930.635,A -85,B 0,C 180,E1 -30230.366,E2 -30230.366} C_VEL
LIN {X 0,Y 37.943,Z 930.563,A -85,B 0,C 180,E1 -30239.995,E2 -30239.995} C_VEL
LIN {X 0,Y 37.282,Z 930.652,A -85,B 0,C 180,E1 -30250.861,E2 -30250.861} C_VEL
LIN {X 0,Y 37.006,Z 930.679,A -85,B 0,C 180,E1 -30258.644,E2 -30258.644} C_VEL
LIN {X 0,Y 35.958,Z 930.81,A -85,B 0,C 180,E1 -30264.529,E2 -30264.529} C_VEL
LIN {X 0,Y 34.202,Z 931.037,A -85,B 0,C 180,E1 -30270.328,E2 -30270.328} C_VEL
LIN {X 0,Y 29.467,Z 931.488,A -85,B 0,C 180,E1 -30291.034,E2 -30291.034} C_VEL
LIN {X 0,Y 29.432,Z 931.461,A -85,B 0,C 180,E1 -30293.719,E2 -30293.719} C_VEL
LIN {X 0,Y 30.306,Z 931.41,A -85,B 0,C 180,E1 -30308.049,E2 -30308.049} C_VEL
LIN {X 0,Y 37.83,Z 930.576,A -85,B 0,C 180,E1 -30340.705,E2 -30340.705} C_VEL
LIN {X 0,Y 43.19,Z 930.016,A -85,B 0,C 180,E1 -30348.222,E2 -30348.222} C_VEL
LIN {X 0,Y 48.369,Z 953.771,A -85,B 0,C 180,E1 -30352.701,E2 -30352.701} C_VEL
LIN {X 0,Y 50.9,Z 964.723,A -85,B 0,C 180,E1 -30354.469,E2 -30354.469} C_VEL
LIN {X 0,Y 55.162,Z 985.868,A -85,B 0,C 180,E1 -30359.845,E2 -30359.845} C_VEL
LIN {X 0,Y 57.392,Z 995.838,A -85,B 0,C 180,E1 -30363.07,E2 -30363.07} C_VEL
LIN {X 0,Y 59.446,Z 1003.029,A -85,B 0,C 180,E1 -30366.235,E2 -30366.235} C_VEL
LIN {X 0,Y 59.988,Z 1005.08,A -85,B 0,C 180,E1 -30367.956,E2 -30367.956} C_VEL
LIN {X 0,Y 61.049,Z 1008.184,A -85,B 0,C 180,E1 -30371.446,E2 -30371.446} C_VEL
LIN {X 0,Y 60.524,Z 1007.234,A -85,B 0,C 180,E1 -30374.163,E2 -30374.163} C_VEL
LIN {X 0,Y 58.064,Z 1000.378,A -85,B 0,C 180,E1 -30379.418,E2 -30379.418} C_VEL
LIN {X 0,Y 56.15,Z 992.828,A -85,B 0,C 180,E1 -30383.803,E2 -30383.803} C_VEL
LIN {X 0,Y 54.328,Z 983.664,A -85,B 0,C 180,E1 -30387.754,E2 -30387.754} C_VEL
LIN {X 0,Y 52.184,Z 972.478,A -85,B 0,C 180,E1 -30391.415,E2 -30391.415} C_VEL
LIN {X 0,Y 45.948,Z 938.158,A -85,B 0,C 180,E1 -30401.223,E2 -30401.223} C_VEL
LIN {X 0,Y 45.023,Z 933.915,A -85,B 0,C 180,E1 -30401.984,E2 -30401.984} C_VEL
LIN {X 0,Y 43.906,Z 929.82,A -85,B 0,C 180,E1 -30402.368,E2 -30402.368} C_VEL
LIN {X 0,Y 38.496,Z 930.5,A -85,B 0,C 180,E1 -30409.486,E2 -30409.486} C_VEL
LIN {X 0,Y 30.211,Z 931.415,A -85,B 0,C 180,E1 -30441.49,E2 -30441.49} C_VEL
LIN {X 0,Y 29.764,Z 931.459,A -85,B 0,C 180,E1 -30448.187,E2 -30448.187} C_VEL
LIN {X 0,Y 29.538,Z 931.482,A -85,B 0,C 180,E1 -30465.554,E2 -30465.554} C_VEL
LIN {X 0,Y 29.471,Z 931.489,A -85,B 0,C 180,E1 -30481.517,E2 -30481.517} C_VEL
LIN {X 0,Y 29.841,Z 931.453,A -85,B 0,C 180,E1 -30490.422,E2 -30490.422} C_VEL
LIN {X 0,Y 30.069,Z 931.429,A -85,B 0,C 180,E1 -30496.486,E2 -30496.486} C_VEL
LIN {X 0,Y 30.768,Z 931.368,A -85,B 0,C 180,E1 -30510.002,E2 -30510.002} C_VEL
LIN {X 0,Y 30.068,Z 931.429,A -85,B 0,C 180,E1 -30523.52,E2 -30523.52} C_VEL
LIN {X 0,Y 29.841,Z 931.453,A -85,B 0,C 180,E1 -30529.58,E2 -30529.58} C_VEL
LIN {X 0,Y 29.472,Z 931.489,A -85,B 0,C 180,E1 -30538.488,E2 -30538.488} C_VEL
LIN {X 0,Y 29.538,Z 931.482,A -85,B 0,C 180,E1 -30555.549,E2 -30555.549} C_VEL
LIN {X 0,Y 29.477,Z 931.486,A -85,B 0,C 180,E1 -30571.513,E2 -30571.513} C_VEL
LIN {X 0,Y 29.84,Z 931.451,A -85,B 0,C 180,E1 -30580.414,E2 -30580.414} C_VEL
LIN {X 0,Y 30.064,Z 931.43,A -85,B 0,C 180,E1 -30586.475,E2 -30586.475} C_VEL
LIN {X 0,Y 30.759,Z 931.365,A -85,B 0,C 180,E1 -30599.994,E2 -30599.994} C_VEL
LIN {X 0,Y 30.071,Z 931.431,A -85,B 0,C 180,E1 -30613.51,E2 -30613.51} C_VEL
LIN {X 0,Y 29.837,Z 931.455,A -85,B 0,C 180,E1 -30619.573,E2 -30619.573} C_VEL
LIN {X 0,Y 29.468,Z 931.488,A -85,B 0,C 180,E1 -30628.482,E2 -30628.482} C_VEL
LIN {X 0,Y 29.585,Z 931.475,A -85,B 0,C 180,E1 -30645.443,E2 -30645.443} C_VEL
LIN {X 0,Y 29.432,Z 931.461,A -85,B 0,C 180,E1 -30653.719,E2 -30653.719} C_VEL
LIN {X 0,Y 29.366,Z 931.496,A -85,B 0,C 180,E1 -30661.336,E2 -30661.336} C_VEL
LIN {X 0,Y 28.919,Z 931.543,A -85,B 0,C 180,E1 -30672.934,E2 -30672.934} C_VEL
LIN {X 0,Y 31.182,Z 931.329,A -85,B 0,C 180,E1 -30703.667,E2 -30703.667} C_VEL
LIN {X 0,Y 34.889,Z 930.927,A -85,B 0,C 180,E1 -30711.846,E2 -30711.846} C_VEL
LIN {X 0,Y 40.286,Z 930.267,A -85,B 0,C 180,E1 -30717.166,E2 -30717.166} C_VEL
LIN {X 0,Y 46.197,Z 954.711,A -85,B 0,C 180,E1 -30720.891,E2 -30720.891} C_VEL
LIN {X 0,Y 48.597,Z 964.375,A -85,B 0,C 180,E1 -30722.226,E2 -30722.226} C_VEL
LIN {X 0,Y 53.355,Z 984.456,A -85,B 0,C 180,E1 -30726.935,E2 -30726.935} C_VEL
LIN {X 0,Y 56.007,Z 994.734,A -85,B 0,C 180,E1 -30730.09,E2 -30730.09} C_VEL
LIN {X 0,Y 56.69,Z 997.166,A -85,B 0,C 180,E1 -30731.094,E2 -30731.094} C_VEL
LIN {X 0,Y 57.083,Z 998.427,A -85,B 0,C 180,E1 -30732.382,E2 -30732.382} C_VEL
LIN {X 0,Y 54.969,Z 992.015,A -85,B 0,C 180,E1 -30736.278,E2 -30736.278} C_VEL
LIN {X 0,Y 52.92,Z 983.769,A -85,B 0,C 180,E1 -30739.927,E2 -30739.927} C_VEL
LIN {X 0,Y 50.42,Z 972.791,A -85,B 0,C 180,E1 -30743.577,E2 -30743.577} C_VEL
LIN {X 0,Y 42.521,Z 936.335,A -85,B 0,C 180,E1 -30753.385,E2 -30753.385} C_VEL
LIN {X 0,Y 40.883,Z 930.193,A -85,B 0,C 180,E1 -30753.687,E2 -30753.687} C_VEL
LIN {X 0,Y 36.609,Z 930.731,A -85,B 0,C 180,E1 -30757.427,E2 -30757.427} C_VEL
LIN {X 0,Y 26.047,Z 931.776,A -85,B 0,C 180,E1 -30780.007,E2 -30780.007} C_VEL
LIN {X 0,Y 22.899,Z 931.875,A -85,B 0,C 180,E1 -30802.976,E2 -30802.976} C_VEL
LIN {X 0,Y 22.287,Z 931.894,A -85,B 0,C 180,E1 -30819.111,E2 -30819.111} C_VEL
LIN {X 0,Y 22.186,Z 931.897,A -85,B 0,C 180,E1 -30830.692,E2 -30830.692} C_VEL
LIN {X 0,Y 22.777,Z 931.879,A -85,B 0,C 180,E1 -30852.031,E2 -30852.031} C_VEL
LIN {X 0,Y 23.542,Z 931.856,A -85,B 0,C 180,E1 -30870.003,E2 -30870.003} C_VEL
LIN {X 0,Y 22.777,Z 931.879,A -85,B 0,C 180,E1 -30887.975,E2 -30887.975} C_VEL
LIN {X 0,Y 22.186,Z 931.897,A -85,B 0,C 180,E1 -30909.316,E2 -30909.316} C_VEL
LIN {X 0,Y 22.188,Z 931.897,A -85,B 0,C 180,E1 -30920.681,E2 -30920.681} C_VEL
LIN {X 0,Y 22.777,Z 931.879,A -85,B 0,C 180,E1 -30942.019,E2 -30942.019} C_VEL
LIN {X 0,Y 23.535,Z 931.856,A -85,B 0,C 180,E1 -30959.992,E2 -30959.992} C_VEL
LIN {X 0,Y 22.774,Z 931.879,A -85,B 0,C 180,E1 -30977.966,E2 -30977.966} C_VEL
LIN {X 0,Y 22.205,Z 931.897,A -85,B 0,C 180,E1 -30999.263,E2 -30999.263} C_VEL
LIN {X 0,Y 22.347,Z 931.888,A -85,B 0,C 180,E1 -31014.104,E2 -31014.104} C_VEL
LIN {X 0,Y 23.466,Z 931.857,A -85,B 0,C 180,E1 -31032.569,E2 -31032.569} C_VEL
LIN {X 0,Y 30.064,Z 931.433,A -85,B 0,C 180,E1 -31063.516,E2 -31063.516} C_VEL
LIN {X 0,Y 34.889,Z 930.927,A -85,B 0,C 180,E1 -31071.846,E2 -31071.846} C_VEL
LIN {X 0,Y 36.756,Z 931.328,A -85,B 0,C 180,E1 -31074.812,E2 -31074.812} C_VEL
LIN {X 0,Y 38.701,Z 933.136,A -85,B 0,C 180,E1 -31078.585,E2 -31078.585} C_VEL
LIN {X 0,Y 40.464,Z 936.656,A -85,B 0,C 180,E1 -31082.648,E2 -31082.648} C_VEL
LIN {X 0,Y 41.704,Z 941.027,A -85,B 0,C 180,E1 -31085.674,E2 -31085.674} C_VEL
LIN {X 0,Y 43.345,Z 948.422,A -85,B 0,C 180,E1 -31088.759,E2 -31088.759} C_VEL
LIN {X 0,Y 45.608,Z 957.142,A -85,B 0,C 180,E1 -31089.867,E2 -31089.867} C_VEL
LIN {X 0,Y 47.573,Z 964.647,A -85,B 0,C 180,E1 -31090.687,E2 -31090.687} C_VEL
LIN {X 0,Y 51.156,Z 978.316,A -85,B 0,C 180,E1 -31093.385,E2 -31093.385} C_VEL
LIN {X 0,Y 51.202,Z 978.512,A -85,B 0,C 180,E1 -31093.643,E2 -31093.643} C_VEL
LIN {X 0,Y 48.5,Z 968.618,A -85,B 0,C 180,E1 -31096.217,E2 -31096.217} C_VEL
LIN {X 0,Y 40.412,Z 935.701,A -85,B 0,C 180,E1 -31104.065,E2 -31104.065} C_VEL
LIN {X 0,Y 38.79,Z 930.453,A -85,B 0,C 180,E1 -31103.931,E2 -31103.931} C_VEL
LIN {X 0,Y 33.544,Z 931.101,A -85,B 0,C 180,E1 -31106.933,E2 -31106.933} C_VEL
LIN {X 0,Y 21.868,Z 931.906,A -85,B 0,C 180,E1 -31124.596,E2 -31124.596} C_VEL
LIN {X 0,Y 18.006,Z 931.991,A -85,B 0,C 180,E1 -31140.01,E2 -31140.01} C_VEL
LIN {X 0,Y 15.381,Z 931.991,A -85,B 0,C 180,E1 -31167.203,E2 -31167.203} C_VEL
LIN {X 0,Y 15.052,Z 931.991,A -85,B 0,C 180,E1 -31202.172,E2 -31202.172} C_VEL
LIN {X 0,Y 15.245,Z 931.991,A -85,B 0,C 180,E1 -31207.258,E2 -31207.258} C_VEL
LIN {X 0,Y 16.216,Z 931.991,A -85,B 0,C 180,E1 -31230.005,E2 -31230.005} C_VEL
LIN {X 0,Y 15.245,Z 931.991,A -85,B 0,C 180,E1 -31252.748,E2 -31252.748} C_VEL
LIN {X 0,Y 15.053,Z 931.991,A -85,B 0,C 180,E1 -31257.839,E2 -31257.839} C_VEL
LIN {X 0,Y 15.053,Z 931.991,A -85,B 0,C 180,E1 -31292.155,E2 -31292.155} C_VEL
LIN {X 0,Y 15.245,Z 931.991,A -85,B 0,C 180,E1 -31297.234,E2 -31297.234} C_VEL
LIN {X 0,Y 16.21,Z 931.991,A -85,B 0,C 180,E1 -31319.988,E2 -31319.988} C_VEL
LIN {X 0,Y 15.244,Z 931.991,A -85,B 0,C 180,E1 -31342.76,E2 -31342.76} C_VEL
LIN {X 0,Y 15.532,Z 931.991,A -85,B 0,C 180,E1 -31383.09,E2 -31383.09} C_VEL
LIN {X 0,Y 17.969,Z 931.991,A -85,B 0,C 180,E1 -31409.996,E2 -31409.996} C_VEL
LIN {X 0,Y 28.63,Z 931.567,A -85,B 0,C 180,E1 -31439.4,E2 -31439.4} C_VEL
LIN {X 0,Y 35.874,Z 930.817,A -85,B 0,C 180,E1 -31445.993,E2 -31445.993} C_VEL
LIN {X 0,Y 38.686,Z 930.465,A -85,B 0,C 180,E1 -31447.199,E2 -31447.199} C_VEL
LIN {X 0,Y 44.594,Z 953.312,A -85,B 0,C 180,E1 -31449.617,E2 -31449.617} C_VEL
LIN {X 0,Y 45.608,Z 957.142,A -85,B 0,C 180,E1 -31449.867,E2 -31449.867} C_VEL
LIN {X 0,Y 44.637,Z 957.032,A -85,B 0,C 180,E1 -31450.336,E2 -31450.336} C_VEL
LIN {X 0,Y 42.96,Z 955.535,A -85,B 0,C 180,E1 -31450.911,E2 -31450.911} C_VEL
LIN {X 0,Y 37.953,Z 948.848,A -85,B 0,C 180,E1 -31452.1,E2 -31452.1} C_VEL
LIN {X 0,Y 34.07,Z 943.2,A -85,B 0,C 180,E1 -31452.603,E2 -31452.603} C_VEL
LIN {X 0,Y 28.793,Z 936.648,A -85,B 0,C 180,E1 -31452.599,E2 -31452.599} C_VEL
LIN {X 0,Y 25.127,Z 933.72,A -85,B 0,C 180,E1 -31451.427,E2 -31451.427} C_VEL
LIN {X 0,Y 21.744,Z 932.216,A -85,B 0,C 180,E1 -31449.022,E2 -31449.022} C_VEL
LIN {X 0,Y 19.662,Z 931.938,A -85,B 0,C 180,E1 -31446.521,E2 -31446.521} C_VEL
LIN {X 0,Y 9.765,Z 931.991,A -85,B 0,C 180,E1 -31409.992,E2 -31409.992} C_VEL
LIN {X 0,Y 7.923,Z 931.991,A -85,B 0,C 180,E1 -31382.447,E2 -31382.447} C_VEL
LIN {X 0,Y 7.797,Z 931.991,A -85,B 0,C 180,E1 -31345.642,E2 -31345.642} C_VEL
LIN {X 0,Y 8.652,Z 931.991,A -85,B 0,C 180,E1 -31319.978,E2 -31319.978} C_VEL
LIN {X 0,Y 7.759,Z 931.991,A -85,B 0,C 180,E1 -31294.96,E2 -31294.96} C_VEL
LIN {X 0,Y 7.759,Z 931.991,A -85,B 0,C 180,E1 -31255.014,E2 -31255.014} C_VEL
LIN {X 0,Y 8.656,Z 931.991,A -85,B 0,C 180,E1 -31230.009,E2 -31230.009} C_VEL
LIN {X 0,Y 7.783,Z 931.991,A -85,B 0,C 180,E1 -31204.606,E2 -31204.606} C_VEL
LIN {X 0,Y 7.872,Z 931.991,A -85,B 0,C 180,E1 -31166.798,E2 -31166.798} C_VEL
LIN {X 0,Y 9.706,Z 931.991,A -85,B 0,C 180,E1 -31140.019,E2 -31140.019} C_VEL
LIN {X 0,Y 22.464,Z 931.889,A -85,B 0,C 180,E1 -31101.276,E2 -31101.276} C_VEL
LIN {X 0,Y 29.274,Z 931.504,A -85,B 0,C 180,E1 -31096.069,E2 -31096.069} C_VEL
LIN {X 0,Y 29.626,Z 931.471,A -85,B 0,C 180,E1 -31095.367,E2 -31095.367} C_VEL
LIN {X 0,Y 19.662,Z 931.938,A -85,B 0,C 180,E1 -31086.521,E2 -31086.521} C_VEL
LIN {X 0,Y 15.118,Z 931.991,A -85,B 0,C 180,E1 -31081.294,E2 -31081.294} C_VEL
LIN {X 0,Y 10.308,Z 931.997,A -85,B 0,C 180,E1 -31077.98,E2 -31077.98} C_VEL
LIN {X 0,Y 0.378,Z 931.991,A -85,B 0,C 180,E1 -31035.215,E2 -31035.215} C_VEL
LIN {X 0,Y 0.307,Z 931.991,A -85,B 0,C 180,E1 -30959.391,E2 -30959.391} C_VEL
LIN {X 0,Y 0.309,Z 931.991,A -85,B 0,C 180,E1 -30870.245,E2 -30870.245} C_VEL
LIN {X 0,Y 0.456,Z 931.991,A -85,B 0,C 180,E1 -30780.41,E2 -30780.41} C_VEL
LIN {X 0,Y 0.378,Z 931.991,A -85,B 0,C 180,E1 -30675.215,E2 -30675.215} C_VEL
LIN {X 0,Y 0.378,Z 931.991,A -85,B 0,C 180,E1 -30675.215,E2 -30675.215}

QRS_NEXT_CUT()

QRS_NEXT()
QRS_HOME()

END
